LIN {X 0,Y 165.753,Z 434.239,A -85,B 0,C 180,E1 -23560.172,E2 -23560.172} C_VEL
LIN {X 0,Y 161.563,Z 431.762,A -85,B 0,C 180,E1 -23564.871,E2 -23564.871} C_VEL
LIN {X 0,Y 158.534,Z 427.948,A -85,B 0,C 180,E1 -23569.786,E2 -23569.786} C_VEL
LIN {X 0,Y 156.538,Z 422.635,A -85,B 0,C 180,E1 -23574.848,E2 -23574.848} C_VEL
LIN {X 0,Y 155.81,Z 417.574,A -85,B 0,C 180,E1 -23578.708,E2 -23578.708} C_VEL
LIN {X 0,Y 155.882,Z 410.304,A -85,B 0,C 180,E1 -23583.231,E2 -23583.231} C_VEL
LIN {X 0,Y 156.223,Z 402.738,A -85,B 0,C 180,E1 -23587.107,E2 -23587.107} C_VEL
LIN {X 0,Y 156.974,Z 393.545,A -85,B 0,C 180,E1 -23590.969,E2 -23590.969} C_VEL
LIN {X 0,Y 158.157,Z 382.372,A -85,B 0,C 180,E1 -23594.804,E2 -23594.804} C_VEL
LIN {X 0,Y 159.494,Z 371.159,A -85,B 0,C 180,E1 -23597.966,E2 -23597.966} C_VEL
LIN {X 0,Y 161.026,Z 358.78,A -85,B 0,C 180,E1 -23600.77,E2 -23600.77} C_VEL
LIN {X 0,Y 161.777,Z 350.482,A -85,B 0,C 180,E1 -23602.342,E2 -23602.342} C_VEL
LIN {X 0,Y 158.681,Z 336.403,A -85,B 0,C 180,E1 -23604.681,E2 -23604.681} C_VEL
LIN {X 0,Y 157.439,Z 330.353,A -85,B 0,C 180,E1 -23605.533,E2 -23605.533} C_VEL
LIN {X 0,Y 157.983,Z 332.419,A -85,B 0,C 180,E1 -23609.298,E2 -23609.298} C_VEL
LIN {X 0,Y 158.474,Z 334.327,A -85,B 0,C 180,E1 -23612.583,E2 -23612.583} C_VEL
LIN {X 0,Y 159.405,Z 337.957,A -85,B 0,C 180,E1 -23618.116,E2 -23618.116} C_VEL
LIN {X 0,Y 159.659,Z 338.968,A -85,B 0,C 180,E1 -23619.459,E2 -23619.459} C_VEL
LIN {X 0,Y 161.445,Z 342.254,A -85,B 0,C 180,E1 -23620.495,E2 -23620.495} C_VEL
LIN {X 0,Y 163.231,Z 344.63,A -85,B 0,C 180,E1 -23621.438,E2 -23621.438} C_VEL
LIN {X 0,Y 166.552,Z 350.082,A -85,B 0,C 180,E1 -23623.291,E2 -23623.291} C_VEL
LIN {X 0,Y 170.558,Z 357.475,A -85,B 0,C 180,E1 -23625.662,E2 -23625.662} C_VEL
LIN {X 0,Y 174.376,Z 366.782,A -85,B 0,C 180,E1 -23628.342,E2 -23628.342} C_VEL
LIN {X 0,Y 176.434,Z 377.226,A -85,B 0,C 180,E1 -23630.963,E2 -23630.963} C_VEL
LIN {X 0,Y 177.459,Z 387.081,A -85,B 0,C 180,E1 -23633.555,E2 -23633.555} C_VEL
LIN {X 0,Y 177.688,Z 393.471,A -85,B 0,C 180,E1 -23635.349,E2 -23635.349} C_VEL
LIN {X 0,Y 177.13,Z 395.819,A -85,B 0,C 180,E1 -23635.914,E2 -23635.914} C_VEL
LIN {X 0,Y 173.857,Z 405.236,A -85,B 0,C 180,E1 -23638.297,E2 -23638.297} C_VEL
LIN {X 0,Y 171.211,Z 412.228,A -85,B 0,C 180,E1 -23640.489,E2 -23640.489} C_VEL
LIN {X 0,Y 167.26,Z 420.911,A -85,B 0,C 180,E1 -23643.82,E2 -23643.82} C_VEL
LIN {X 0,Y 163.998,Z 427.85,A -85,B 0,C 180,E1 -23647.313,E2 -23647.313} C_VEL
LIN {X 0,Y 161.206,Z 433.361,A -85,B 0,C 180,E1 -23650.915,E2 -23650.915} C_VEL
LIN {X 0,Y 158.948,Z 437.681,A -85,B 0,C 180,E1 -23654.615,E2 -23654.615} C_VEL
LIN {X 0,Y 157.815,Z 439.949,A -85,B 0,C 180,E1 -23657.134,E2 -23657.134} C_VEL
LIN {X 0,Y 156.561,Z 442.532,A -85,B 0,C 180,E1 -23660.962,E2 -23660.962} C_VEL
LIN {X 0,Y 155.775,Z 444.181,A -85,B 0,C 180,E1 -23664.823,E2 -23664.823} C_VEL
LIN {X 0,Y 155.382,Z 445.015,A -85,B 0,C 180,E1 -23670,E2 -23670} C_VEL
LIN {X 0,Y 155.466,Z 444.818,A -85,B 0,C 180,E1 -23672.591,E2 -23672.591} C_VEL
LIN {X 0,Y 156.224,Z 443.266,A -85,B 0,C 180,E1 -23677.756,E2 -23677.756} C_VEL
LIN {X 0,Y 156.889,Z 441.903,A -85,B 0,C 180,E1 -23680.322,E2 -23680.322} C_VEL
LIN {X 0,Y 158.282,Z 439.04,A -85,B 0,C 180,E1 -23684.135,E2 -23684.135} C_VEL
LIN {X 0,Y 160.319,Z 435.137,A -85,B 0,C 180,E1 -23687.87,E2 -23687.87} C_VEL
LIN {X 0,Y 162.92,Z 430.072,A -85,B 0,C 180,E1 -23691.511,E2 -23691.511} C_VEL
LIN {X 0,Y 165.997,Z 423.682,A -85,B 0,C 180,E1 -23695.048,E2 -23695.048} C_VEL
LIN {X 0,Y 169.805,Z 415.717,A -85,B 0,C 180,E1 -23698.423,E2 -23698.423} C_VEL
LIN {X 0,Y 173.186,Z 407.595,A -85,B 0,C 180,E1 -23701.15,E2 -23701.15} C_VEL
LIN {X 0,Y 176.252,Z 398.682,A -85,B 0,C 180,E1 -23703.591,E2 -23703.591} C_VEL
LIN {X 0,Y 177.751,Z 394.094,A -85,B 0,C 180,E1 -23704.637,E2 -23704.637} C_VEL
LIN {X 0,Y 177.274,Z 383.59,A -85,B 0,C 180,E1 -23707.542,E2 -23707.542} C_VEL
LIN {X 0,Y 175.939,Z 373.719,A -85,B 0,C 180,E1 -23710.085,E2 -23710.085} C_VEL
LIN {X 0,Y 174.068,Z 365.643,A -85,B 0,C 180,E1 -23712.143,E2 -23712.143} C_VEL
LIN {X 0,Y 170.123,Z 356.525,A -85,B 0,C 180,E1 -23714.824,E2 -23714.824} C_VEL
LIN {X 0,Y 165.27,Z 347.901,A -85,B 0,C 180,E1 -23717.637,E2 -23717.637} C_VEL
LIN {X 0,Y 162.421,Z 343.392,A -85,B 0,C 180,E1 -23719.218,E2 -23719.218} C_VEL
LIN {X 0,Y 160.135,Z 340.062,A -85,B 0,C 180,E1 -23720.478,E2 -23720.478} C_VEL
LIN {X 0,Y 159.646,Z 338.902,A -85,B 0,C 180,E1 -23720.873,E2 -23720.873} C_VEL
LIN {X 0,Y 158.84,Z 336.211,A -85,B 0,C 180,E1 -23724.887,E2 -23724.887} C_VEL
LIN {X 0,Y 157.779,Z 334.62,A -85,B 0,C 180,E1 -23727.815,E2 -23727.815} C_VEL
LIN {X 0,Y 156.887,Z 333.987,A -85,B 0,C 180,E1 -23729.706,E2 -23729.706} C_VEL
LIN {X 0,Y 156.589,Z 338.43,A -85,B 0,C 180,E1 -23733.887,E2 -23733.887} C_VEL
LIN {X 0,Y 158.408,Z 353.582,A -85,B 0,C 180,E1 -23735.786,E2 -23735.786} C_VEL
LIN {X 0,Y 160.641,Z 367.663,A -85,B 0,C 180,E1 -23738.039,E2 -23738.039} C_VEL
LIN {X 0,Y 160.973,Z 370.884,A -85,B 0,C 180,E1 -23738.627,E2 -23738.627} C_VEL
LIN {X 0,Y 159.654,Z 382.742,A -85,B 0,C 180,E1 -23741.055,E2 -23741.055} C_VEL
LIN {X 0,Y 158.31,Z 393.87,A -85,B 0,C 180,E1 -23743.891,E2 -23743.891} C_VEL
LIN {X 0,Y 157.104,Z 404.147,A -85,B 0,C 180,E1 -23747.075,E2 -23747.075} C_VEL
LIN {X 0,Y 156.285,Z 412.837,A -85,B 0,C 180,E1 -23750.291,E2 -23750.291} C_VEL
LIN {X 0,Y 155.643,Z 421.458,A -85,B 0,C 180,E1 -23754.151,E2 -23754.151} C_VEL
LIN {X 0,Y 155.47,Z 428.59,A -85,B 0,C 180,E1 -23758.057,E2 -23758.057} C_VEL
LIN {X 0,Y 155.577,Z 435.33,A -85,B 0,C 180,E1 -23762.589,E2 -23762.589} C_VEL
LIN {X 0,Y 156.239,Z 439.911,A -85,B 0,C 180,E1 -23766.457,E2 -23766.457} C_VEL
LIN {X 0,Y 157.731,Z 444.459,A -85,B 0,C 180,E1 -23771.404,E2 -23771.404} C_VEL
LIN {X 0,Y 159.963,Z 447.144,A -85,B 0,C 180,E1 -23775.284,E2 -23775.284} C_VEL
LIN {X 0,Y 163.92,Z 449.371,A -85,B 0,C 180,E1 -23780.06,E2 -23780.06} C_VEL
LIN {X 0,Y 169.127,Z 450.293,A -85,B 0,C 180,E1 -23784.554,E2 -23784.554} C_VEL
LIN {X 0,Y 175.467,Z 449.904,A -85,B 0,C 180,E1 -23788.727,E2 -23788.727} C_VEL
LIN {X 0,Y 182.919,Z 448.24,A -85,B 0,C 180,E1 -23792.541,E2 -23792.541} C_VEL
LIN {X 0,Y 191.342,Z 445.326,A -85,B 0,C 180,E1 -23795.993,E2 -23795.993} C_VEL
LIN {X 0,Y 200.7,Z 441.045,A -85,B 0,C 180,E1 -23799.073,E2 -23799.073} C_VEL
LIN {X 0,Y 210.694,Z 435.47,A -85,B 0,C 180,E1 -23801.846,E2 -23801.846} C_VEL
LIN {X 0,Y 211.205,Z 435.279,A -85,B 0,C 180,E1 -23802.94,E2 -23802.94} C_VEL
LIN {X 0,Y 210.36,Z 436.026,A -85,B 0,C 180,E1 -23804.085,E2 -23804.085} C_VEL
LIN {X 0,Y 206.003,Z 439.07,A -85,B 0,C 180,E1 -23805.623,E2 -23805.623} C_VEL
LIN {X 0,Y 194.505,Z 446.435,A -85,B 0,C 180,E1 -23809.429,E2 -23809.429} C_VEL
LIN {X 0,Y 185.399,Z 451.418,A -85,B 0,C 180,E1 -23812.662,E2 -23812.662} C_VEL
LIN {X 0,Y 177.209,Z 455.306,A -85,B 0,C 180,E1 -23816.273,E2 -23816.273} C_VEL
LIN {X 0,Y 170.283,Z 458.104,A -85,B 0,C 180,E1 -23820.312,E2 -23820.312} C_VEL
LIN {X 0,Y 164.595,Z 459.85,A -85,B 0,C 180,E1 -23824.723,E2 -23824.723} C_VEL
LIN {X 0,Y 160.207,Z 460.514,A -85,B 0,C 180,E1 -23829.455,E2 -23829.455} C_VEL
LIN {X 0,Y 157.293,Z 460.078,A -85,B 0,C 180,E1 -23834.45,E2 -23834.45} C_VEL
LIN {X 0,Y 156.148,Z 459.074,A -85,B 0,C 180,E1 -23838.479,E2 -23838.479} C_VEL
LIN {X 0,Y 155.39,Z 461.312,A -85,B 0,C 180,E1 -23842.202,E2 -23842.202} C_VEL
LIN {X 0,Y 155.146,Z 462.974,A -85,B 0,C 180,E1 -23847.404,E2 -23847.404} C_VEL
LIN {X 0,Y 155.383,Z 463.209,A -85,B 0,C 180,E1 -23850,E2 -23850} C_VEL
LIN {X 0,Y 155.08,Z 462.56,A -85,B 0,C 180,E1 -23854.433,E2 -23854.433} C_VEL
LIN {X 0,Y 155.153,Z 461.271,A -85,B 0,C 180,E1 -23857.81,E2 -23857.81} C_VEL
LIN {X 0,Y 155.501,Z 459.802,A -85,B 0,C 180,E1 -23860.415,E2 -23860.415} C_VEL
LIN {X 0,Y 156.455,Z 456.851,A -85,B 0,C 180,E1 -23864.204,E2 -23864.204} C_VEL
LIN {X 0,Y 156.313,Z 455.572,A -85,B 0,C 180,E1 -23865.589,E2 -23865.589} C_VEL
LIN {X 0,Y 153.093,Z 451.08,A -85,B 0,C 180,E1 -23870.172,E2 -23870.172} C_VEL
LIN {X 0,Y 153.396,Z 450.467,A -85,B 0,C 180,E1 -23871.636,E2 -23871.636} C_VEL
LIN {X 0,Y 157.584,Z 449.759,A -85,B 0,C 180,E1 -23876.486,E2 -23876.486} C_VEL
LIN {X 0,Y 163.273,Z 448.055,A -85,B 0,C 180,E1 -23881.1,E2 -23881.1} C_VEL
LIN {X 0,Y 170.372,Z 445.383,A -85,B 0,C 180,E1 -23885.276,E2 -23885.276} C_VEL
LIN {X 0,Y 178.668,Z 441.731,A -85,B 0,C 180,E1 -23889.004,E2 -23889.004} C_VEL
LIN {X 0,Y 189.566,Z 435.946,A -85,B 0,C 180,E1 -23893.305,E2 -23893.305} C_VEL
LIN {X 0,Y 193.556,Z 433.494,A -85,B 0,C 180,E1 -23895.076,E2 -23895.076} C_VEL
LIN {X 0,Y 195.412,Z 432.26,A -85,B 0,C 180,E1 -23895.997,E2 -23895.997} C_VEL
LIN {X 0,Y 197.524,Z 430.74,A -85,B 0,C 180,E1 -23897.466,E2 -23897.466} C_VEL
LIN {X 0,Y 197.825,Z 430.354,A -85,B 0,C 180,E1 -23898.25,E2 -23898.25} C_VEL
LIN {X 0,Y 198.082,Z 429.735,A -85,B 0,C 180,E1 -23900.309,E2 -23900.309} C_VEL
LIN {X 0,Y 188.461,Z 433.218,A -85,B 0,C 180,E1 -23903.369,E2 -23903.369} C_VEL
LIN {X 0,Y 179.669,Z 435.441,A -85,B 0,C 180,E1 -23906.796,E2 -23906.796} C_VEL
LIN {X 0,Y 171.721,Z 436.42,A -85,B 0,C 180,E1 -23910.586,E2 -23910.586} C_VEL
LIN {X 0,Y 164.78,Z 436.179,A -85,B 0,C 180,E1 -23914.754,E2 -23914.754} C_VEL
LIN {X 0,Y 159.11,Z 434.652,A -85,B 0,C 180,E1 -23919.307,E2 -23919.307} C_VEL
LIN {X 0,Y 154.737,Z 431.839,A -85,B 0,C 180,E1 -23924.186,E2 -23924.186} C_VEL
LIN {X 0,Y 151.567,Z 427.625,A -85,B 0,C 180,E1 -23929.311,E2 -23929.311} C_VEL
LIN {X 0,Y 149.492,Z 421.939,A -85,B 0,C 180,E1 -23934.605,E2 -23934.605} C_VEL
LIN {X 0,Y 148.727,Z 414.582,A -85,B 0,C 180,E1 -23940,E2 -23940} C_VEL
LIN {X 0,Y 149.03,Z 406.5,A -85,B 0,C 180,E1 -23944.734,E2 -23944.734} C_VEL
LIN {X 0,Y 149.553,Z 396.83,A -85,B 0,C 180,E1 -23949.297,E2 -23949.297} C_VEL
LIN {X 0,Y 150.411,Z 387.773,A -85,B 0,C 180,E1 -23952.824,E2 -23952.824} C_VEL
LIN {X 0,Y 151.711,Z 376.334,A -85,B 0,C 180,E1 -23956.484,E2 -23956.484} C_VEL
LIN {X 0,Y 153.302,Z 363.69,A -85,B 0,C 180,E1 -23959.761,E2 -23959.761} C_VEL
LIN {X 0,Y 154.707,Z 352.272,A -85,B 0,C 180,E1 -23962.167,E2 -23962.167} C_VEL
LIN {X 0,Y 152.905,Z 343.422,A -85,B 0,C 180,E1 -23963.779,E2 -23963.779} C_VEL
LIN {X 0,Y 150.839,Z 333.597,A -85,B 0,C 180,E1 -23965.402,E2 -23965.402} C_VEL
LIN {X 0,Y 151.352,Z 334.822,A -85,B 0,C 180,E1 -23968.083,E2 -23968.083} C_VEL
LIN {X 0,Y 152.138,Z 337.991,A -85,B 0,C 180,E1 -23973.746,E2 -23973.746} C_VEL
LIN {X 0,Y 152.527,Z 339.479,A -85,B 0,C 180,E1 -23976.08,E2 -23976.08} C_VEL
LIN {X 0,Y 154.477,Z 342.78,A -85,B 0,C 180,E1 -23977.367,E2 -23977.367} C_VEL
LIN {X 0,Y 156.395,Z 345.088,A -85,B 0,C 180,E1 -23978.51,E2 -23978.51} C_VEL
LIN {X 0,Y 158.911,Z 349.057,A -85,B 0,C 180,E1 -23980.094,E2 -23980.094} C_VEL
LIN {X 0,Y 162.644,Z 355.633,A -85,B 0,C 180,E1 -23982.5,E2 -23982.5} C_VEL
LIN {X 0,Y 166.311,Z 363.122,A -85,B 0,C 180,E1 -23985.059,E2 -23985.059} C_VEL
LIN {X 0,Y 169.218,Z 370.991,A -85,B 0,C 180,E1 -23987.494,E2 -23987.494} C_VEL
LIN {X 0,Y 170.838,Z 380.954,A -85,B 0,C 180,E1 -23990.188,E2 -23990.188} C_VEL
LIN {X 0,Y 171.504,Z 390.512,A -85,B 0,C 180,E1 -23992.898,E2 -23992.898} C_VEL
LIN {X 0,Y 171.539,Z 395.184,A -85,B 0,C 180,E1 -23994.308,E2 -23994.308} C_VEL
LIN {X 0,Y 167.86,Z 405.647,A -85,B 0,C 180,E1 -23997.024,E2 -23997.024} C_VEL
LIN {X 0,Y 165.094,Z 412.639,A -85,B 0,C 180,E1 -23999.28,E2 -23999.28} C_VEL
LIN {X 0,Y 160.935,Z 421.324,A -85,B 0,C 180,E1 -24002.707,E2 -24002.707} C_VEL
LIN {X 0,Y 157.48,Z 428.265,A -85,B 0,C 180,E1 -24006.318,E2 -24006.318} C_VEL
LIN {X 0,Y 154.521,Z 433.776,A -85,B 0,C 180,E1 -24010.055,E2 -24010.055} C_VEL
LIN {X 0,Y 152.12,Z 438.097,A -85,B 0,C 180,E1 -24013.907,E2 -24013.907} C_VEL
LIN {X 0,Y 150.921,Z 440.363,A -85,B 0,C 180,E1 -24016.536,E2 -24016.536} C_VEL
LIN {X 0,Y 149.496,Z 443.105,A -85,B 0,C 180,E1 -24020.838,E2 -24020.838} C_VEL
LIN {X 0,Y 148.726,Z 444.595,A -85,B 0,C 180,E1 -24024.577,E2 -24024.577} C_VEL
LIN {X 0,Y 148.301,Z 445.43,A -85,B 0,C 180,E1 -24030,E2 -24030} C_VEL
LIN {X 0,Y 148.393,Z 445.232,A -85,B 0,C 180,E1 -24032.715,E2 -24032.715} C_VEL
LIN {X 0,Y 149.215,Z 443.68,A -85,B 0,C 180,E1 -24038.123,E2 -24038.123} C_VEL
LIN {X 0,Y 149.915,Z 442.318,A -85,B 0,C 180,E1 -24040.808,E2 -24040.808} C_VEL
LIN {X 0,Y 151.425,Z 439.453,A -85,B 0,C 180,E1 -24044.79,E2 -24044.79} C_VEL
LIN {X 0,Y 153.582,Z 435.55,A -85,B 0,C 180,E1 -24048.683,E2 -24048.683} C_VEL
LIN {X 0,Y 156.353,Z 430.482,A -85,B 0,C 180,E1 -24052.462,E2 -24052.462} C_VEL
LIN {X 0,Y 159.6,Z 424.092,A -85,B 0,C 180,E1 -24056.126,E2 -24056.126} C_VEL
LIN {X 0,Y 163.622,Z 416.123,A -85,B 0,C 180,E1 -24059.601,E2 -24059.601} C_VEL
LIN {X 0,Y 167.108,Z 408.095,A -85,B 0,C 180,E1 -24062.379,E2 -24062.379} C_VEL
LIN {X 0,Y 170.363,Z 399.191,A -85,B 0,C 180,E1 -24064.881,E2 -24064.881} C_VEL
LIN {X 0,Y 171.58,Z 395.68,A -85,B 0,C 180,E1 -24065.704,E2 -24065.704} C_VEL
LIN {X 0,Y 171.41,Z 386.763,A -85,B 0,C 180,E1 -24068.346,E2 -24068.346} C_VEL
LIN {X 0,Y 170.239,Z 375.936,A -85,B 0,C 180,E1 -24071.341,E2 -24071.341} C_VEL
LIN {X 0,Y 168.776,Z 369.321,A -85,B 0,C 180,E1 -24073.167,E2 -24073.167} C_VEL
LIN {X 0,Y 165.587,Z 361.345,A -85,B 0,C 180,E1 -24075.718,E2 -24075.718} C_VEL
LIN {X 0,Y 161.339,Z 353.166,A -85,B 0,C 180,E1 -24078.58,E2 -24078.58} C_VEL
LIN {X 0,Y 158.362,Z 348.322,A -85,B 0,C 180,E1 -24080.463,E2 -24080.463} C_VEL
LIN {X 0,Y 155.848,Z 344.352,A -85,B 0,C 180,E1 -24082.055,E2 -24082.055} C_VEL
LIN {X 0,Y 152.98,Z 340.619,A -85,B 0,C 180,E1 -24083.839,E2 -24083.839} C_VEL
LIN {X 0,Y 152.449,Z 339.441,A -85,B 0,C 180,E1 -24084.305,E2 -24084.305} C_VEL
LIN {X 0,Y 151.762,Z 338.268,A -85,B 0,C 180,E1 -24086.468,E2 -24086.468} C_VEL
LIN {X 0,Y 150.617,Z 337.054,A -85,B 0,C 180,E1 -24089.117,E2 -24089.117} C_VEL
LIN {X 0,Y 149.674,Z 336.321,A -85,B 0,C 180,E1 -24091.23,E2 -24091.23} C_VEL
LIN {X 0,Y 149.517,Z 338.899,A -85,B 0,C 180,E1 -24093.734,E2 -24093.734} C_VEL
LIN {X 0,Y 151.314,Z 354.037,A -85,B 0,C 180,E1 -24095.692,E2 -24095.692} C_VEL
LIN {X 0,Y 153.57,Z 368.285,A -85,B 0,C 180,E1 -24098.077,E2 -24098.077} C_VEL
LIN {X 0,Y 153.869,Z 370.852,A -85,B 0,C 180,E1 -24098.567,E2 -24098.567} C_VEL
LIN {X 0,Y 152.513,Z 382.915,A -85,B 0,C 180,E1 -24101.181,E2 -24101.181} C_VEL
LIN {X 0,Y 151,Z 395.136,A -85,B 0,C 180,E1 -24104.477,E2 -24104.477} C_VEL
LIN {X 0,Y 149.868,Z 405.309,A -85,B 0,C 180,E1 -24107.817,E2 -24107.817} C_VEL
LIN {X 0,Y 149.094,Z 413.784,A -85,B 0,C 180,E1 -24111.188,E2 -24111.188} C_VEL
LIN {X 0,Y 148.566,Z 422.244,A -85,B 0,C 180,E1 -24115.251,E2 -24115.251} C_VEL
LIN {X 0,Y 148.463,Z 429.301,A -85,B 0,C 180,E1 -24119.322,E2 -24119.322} C_VEL
LIN {X 0,Y 148.76,Z 435.899,A -85,B 0,C 180,E1 -24124.064,E2 -24124.064} C_VEL
LIN {X 0,Y 149.57,Z 440.46,A -85,B 0,C 180,E1 -24128.104,E2 -24128.104} C_VEL
LIN {X 0,Y 151.519,Z 445.084,A -85,B 0,C 180,E1 -24133.41,E2 -24133.41} C_VEL
LIN {X 0,Y 155.053,Z 448.373,A -85,B 0,C 180,E1 -24138.499,E2 -24138.499} C_VEL
LIN {X 0,Y 159.788,Z 450.348,A -85,B 0,C 180,E1 -24143.319,E2 -24143.319} C_VEL
LIN {X 0,Y 165.848,Z 451,A -85,B 0,C 180,E1 -24147.784,E2 -24147.784} C_VEL
LIN {X 0,Y 173.102,Z 450.409,A -85,B 0,C 180,E1 -24151.857,E2 -24151.857} C_VEL
LIN {X 0,Y 181.833,Z 448.487,A -85,B 0,C 180,E1 -24155.74,E2 -24155.74} C_VEL
LIN {X 0,Y 190.575,Z 445.528,A -85,B 0,C 180,E1 -24158.824,E2 -24158.824} C_VEL
LIN {X 0,Y 200.582,Z 441.177,A -85,B 0,C 180,E1 -24161.738,E2 -24161.738} C_VEL
LIN {X 0,Y 204.307,Z 439.31,A -85,B 0,C 180,E1 -24162.7,E2 -24162.7} C_VEL
LIN {X 0,Y 203.582,Z 439.873,A -85,B 0,C 180,E1 -24163.534,E2 -24163.534} C_VEL
LIN {X 0,Y 191.618,Z 446.746,A -85,B 0,C 180,E1 -24167.271,E2 -24167.271} C_VEL
LIN {X 0,Y 183.001,Z 451.032,A -85,B 0,C 180,E1 -24170.182,E2 -24170.182} C_VEL
LIN {X 0,Y 175.486,Z 454.225,A -85,B 0,C 180,E1 -24173.077,E2 -24173.077} C_VEL
LIN {X 0,Y 167.006,Z 457.295,A -85,B 0,C 180,E1 -24177.315,E2 -24177.315} C_VEL
LIN {X 0,Y 161.028,Z 458.939,A -85,B 0,C 180,E1 -24181.309,E2 -24181.309} C_VEL
LIN {X 0,Y 155.691,Z 459.759,A -85,B 0,C 180,E1 -24186.029,E2 -24186.029} C_VEL
LIN {X 0,Y 151.805,Z 459.525,A -85,B 0,C 180,E1 -24191.09,E2 -24191.09} C_VEL
LIN {X 0,Y 149.455,Z 458.077,A -85,B 0,C 180,E1 -24197.093,E2 -24197.093} C_VEL
LIN {X 0,Y 148.349,Z 460.897,A -85,B 0,C 180,E1 -24201.829,E2 -24201.829} C_VEL
LIN {X 0,Y 148.068,Z 462.178,A -85,B 0,C 180,E1 -24205.387,E2 -24205.387} C_VEL
LIN {X 0,Y 148.29,Z 462.794,A -85,B 0,C 180,E1 -24210,E2 -24210} C_VEL
LIN {X 0,Y 148.01,Z 462.237,A -85,B 0,C 180,E1 -24214.328,E2 -24214.328} C_VEL
LIN {X 0,Y 148.084,Z 460.853,A -85,B 0,C 180,E1 -24218.186,E2 -24218.186} C_VEL
LIN {X 0,Y 148.497,Z 459.384,A -85,B 0,C 180,E1 -24220.913,E2 -24220.913} C_VEL
LIN {X 0,Y 149.591,Z 456.351,A -85,B 0,C 180,E1 -24224.975,E2 -24224.975} C_VEL
LIN {X 0,Y 151.576,Z 452.267,A -85,B 0,C 180,E1 -24228.939,E2 -24228.939} C_VEL
LIN {X 0,Y 152.564,Z 450.503,A -85,B 0,C 180,E1 -24230.388,E2 -24230.388} C_VEL
LIN {X 0,Y 153.396,Z 450.467,A -85,B 0,C 180,E1 -24231.636,E2 -24231.636} C_VEL
LIN {X 0,Y 154.375,Z 450.218,A -85,B 0,C 180,E1 -24233.806,E2 -24233.806} C_VEL
LIN {X 0,Y 155.587,Z 448.449,A -85,B 0,C 180,E1 -24240.363,E2 -24240.363} C_VEL
LIN {X 0,Y 157.292,Z 447.668,A -85,B 0,C 180,E1 -24242.407,E2 -24242.407} C_VEL
LIN {X 0,Y 158.172,Z 447.386,A -85,B 0,C 180,E1 -24243.036,E2 -24243.036} C_VEL
LIN {X 0,Y 164.638,Z 445.411,A -85,B 0,C 180,E1 -24246.7,E2 -24246.7} C_VEL
LIN {X 0,Y 173.226,Z 442.231,A -85,B 0,C 180,E1 -24250.477,E2 -24250.477} C_VEL
LIN {X 0,Y 184.514,Z 437.059,A -85,B 0,C 180,E1 -24254.802,E2 -24254.802} C_VEL
LIN {X 0,Y 188.637,Z 434.859,A -85,B 0,C 180,E1 -24256.595,E2 -24256.595} C_VEL
LIN {X 0,Y 190.392,Z 433.799,A -85,B 0,C 180,E1 -24257.584,E2 -24257.584} C_VEL
LIN {X 0,Y 191.359,Z 433.091,A -85,B 0,C 180,E1 -24258.617,E2 -24258.617} C_VEL
LIN {X 0,Y 190.438,Z 433.174,A -85,B 0,C 180,E1 -24259.772,E2 -24259.772} C_VEL
LIN {X 0,Y 183.02,Z 435.254,A -85,B 0,C 180,E1 -24262.091,E2 -24262.091} C_VEL
LIN {X 0,Y 173.918,Z 436.996,A -85,B 0,C 180,E1 -24265.546,E2 -24265.546} C_VEL
LIN {X 0,Y 165.647,Z 437.572,A -85,B 0,C 180,E1 -24269.394,E2 -24269.394} C_VEL
LIN {X 0,Y 158.429,Z 436.887,A -85,B 0,C 180,E1 -24273.666,E2 -24273.666} C_VEL
LIN {X 0,Y 152.509,Z 434.941,A -85,B 0,C 180,E1 -24278.367,E2 -24278.367} C_VEL
LIN {X 0,Y 147.938,Z 431.727,A -85,B 0,C 180,E1 -24283.439,E2 -24283.439} C_VEL
LIN {X 0,Y 144.614,Z 427.179,A -85,B 0,C 180,E1 -24288.791,E2 -24288.791} C_VEL
LIN {X 0,Y 142.462,Z 421.11,A -85,B 0,C 180,E1 -24294.338,E2 -24294.338} C_VEL
LIN {X 0,Y 141.71,Z 413.335,A -85,B 0,C 180,E1 -24300,E2 -24300} C_VEL
LIN {X 0,Y 142.023,Z 404.891,A -85,B 0,C 180,E1 -24304.968,E2 -24304.968} C_VEL
LIN {X 0,Y 142.529,Z 395.794,A -85,B 0,C 180,E1 -24309.293,E2 -24309.293} C_VEL
LIN {X 0,Y 143.579,Z 385.207,A -85,B 0,C 180,E1 -24313.445,E2 -24313.445} C_VEL
LIN {X 0,Y 144.969,Z 373.249,A -85,B 0,C 180,E1 -24317.274,E2 -24317.274} C_VEL
LIN {X 0,Y 146.487,Z 361.182,A -85,B 0,C 180,E1 -24320.355,E2 -24320.355} C_VEL
LIN {X 0,Y 147.48,Z 353.393,A -85,B 0,C 180,E1 -24322.042,E2 -24322.042} C_VEL
LIN {X 0,Y 147.488,Z 351.505,A -85,B 0,C 180,E1 -24322.409,E2 -24322.409} C_VEL
LIN {X 0,Y 144.535,Z 338.06,A -85,B 0,C 180,E1 -24324.854,E2 -24324.854} C_VEL
LIN {X 0,Y 144.246,Z 336.748,A -85,B 0,C 180,E1 -24325.127,E2 -24325.127} C_VEL
LIN {X 0,Y 144.643,Z 336.965,A -85,B 0,C 180,E1 -24325.932,E2 -24325.932} C_VEL
LIN {X 0,Y 145.352,Z 339.638,A -85,B 0,C 180,E1 -24331.317,E2 -24331.317} C_VEL
LIN {X 0,Y 145.559,Z 340.272,A -85,B 0,C 180,E1 -24332.149,E2 -24332.149} C_VEL
LIN {X 0,Y 147.748,Z 343.714,A -85,B 0,C 180,E1 -24333.845,E2 -24333.845} C_VEL
LIN {X 0,Y 149.613,Z 345.751,A -85,B 0,C 180,E1 -24335.131,E2 -24335.131} C_VEL
LIN {X 0,Y 152.192,Z 349.675,A -85,B 0,C 180,E1 -24336.997,E2 -24336.997} C_VEL
LIN {X 0,Y 156.002,Z 356.166,A -85,B 0,C 180,E1 -24339.765,E2 -24339.765} C_VEL
LIN {X 0,Y 158.485,Z 360.883,A -85,B 0,C 180,E1 -24341.638,E2 -24341.638} C_VEL
LIN {X 0,Y 161.539,Z 367.596,A -85,B 0,C 180,E1 -24344.116,E2 -24344.116} C_VEL
LIN {X 0,Y 163.836,Z 374.444,A -85,B 0,C 180,E1 -24346.422,E2 -24346.422} C_VEL
LIN {X 0,Y 165.028,Z 383.315,A -85,B 0,C 180,E1 -24349.002,E2 -24349.002} C_VEL
LIN {X 0,Y 165.477,Z 392.709,A -85,B 0,C 180,E1 -24351.86,E2 -24351.86} C_VEL
LIN {X 0,Y 165.46,Z 395.829,A -85,B 0,C 180,E1 -24352.854,E2 -24352.854} C_VEL
LIN {X 0,Y 164.733,Z 398.923,A -85,B 0,C 180,E1 -24353.705,E2 -24353.705} C_VEL
LIN {X 0,Y 161.579,Z 407.086,A -85,B 0,C 180,E1 -24355.975,E2 -24355.975} C_VEL
LIN {X 0,Y 158.273,Z 414.645,A -85,B 0,C 180,E1 -24358.55,E2 -24358.55} C_VEL
LIN {X 0,Y 154.681,Z 421.737,A -85,B 0,C 180,E1 -24361.505,E2 -24361.505} C_VEL
LIN {X 0,Y 151.025,Z 428.678,A -85,B 0,C 180,E1 -24365.24,E2 -24365.24} C_VEL
LIN {X 0,Y 147.867,Z 434.192,A -85,B 0,C 180,E1 -24369.116,E2 -24369.116} C_VEL
LIN {X 0,Y 145.33,Z 438.511,A -85,B 0,C 180,E1 -24373.133,E2 -24373.133} C_VEL
LIN {X 0,Y 144.024,Z 440.779,A -85,B 0,C 180,E1 -24375.878,E2 -24375.878} C_VEL
LIN {X 0,Y 142.376,Z 443.75,A -85,B 0,C 180,E1 -24380.841,E2 -24380.841} C_VEL
LIN {X 0,Y 141.681,Z 445.01,A -85,B 0,C 180,E1 -24384.306,E2 -24384.306} C_VEL
LIN {X 0,Y 141.221,Z 445.844,A -85,B 0,C 180,E1 -24390,E2 -24390} C_VEL
LIN {X 0,Y 141.322,Z 445.646,A -85,B 0,C 180,E1 -24392.851,E2 -24392.851} C_VEL
LIN {X 0,Y 141.658,Z 445.059,A -85,B 0,C 180,E1 -24395.695,E2 -24395.695} C_VEL
LIN {X 0,Y 142.32,Z 443.9,A -85,B 0,C 180,E1 -24399.018,E2 -24399.018} C_VEL
LIN {X 0,Y 143.972,Z 440.909,A -85,B 0,C 180,E1 -24404.127,E2 -24404.127} C_VEL
LIN {X 0,Y 146.041,Z 437.362,A -85,B 0,C 180,E1 -24408.228,E2 -24408.228} C_VEL
LIN {X 0,Y 148.809,Z 432.697,A -85,B 0,C 180,E1 -24412.199,E2 -24412.199} C_VEL
LIN {X 0,Y 152.094,Z 426.782,A -85,B 0,C 180,E1 -24416.039,E2 -24416.039} C_VEL
LIN {X 0,Y 156.014,Z 419.406,A -85,B 0,C 180,E1 -24419.704,E2 -24419.704} C_VEL
LIN {X 0,Y 160.277,Z 410.568,A -85,B 0,C 180,E1 -24423.046,E2 -24423.046} C_VEL
LIN {X 0,Y 164.15,Z 400.747,A -85,B 0,C 180,E1 -24425.989,E2 -24425.989} C_VEL
LIN {X 0,Y 165.447,Z 397.325,A -85,B 0,C 180,E1 -24426.83,E2 -24426.83} C_VEL
LIN {X 0,Y 165.483,Z 388.614,A -85,B 0,C 180,E1 -24429.572,E2 -24429.572} C_VEL
LIN {X 0,Y 164.566,Z 378.245,A -85,B 0,C 180,E1 -24432.641,E2 -24432.641} C_VEL
LIN {X 0,Y 163.095,Z 371.63,A -85,B 0,C 180,E1 -24434.683,E2 -24434.683} C_VEL
LIN {X 0,Y 159.337,Z 362.386,A -85,B 0,C 180,E1 -24437.969,E2 -24437.969} C_VEL
LIN {X 0,Y 154.999,Z 354.231,A -85,B 0,C 180,E1 -24441.223,E2 -24441.223} C_VEL
LIN {X 0,Y 152.226,Z 349.783,A -85,B 0,C 180,E1 -24443.22,E2 -24443.22} C_VEL
LIN {X 0,Y 149.553,Z 345.761,A -85,B 0,C 180,E1 -24445.161,E2 -24445.161} C_VEL
LIN {X 0,Y 144.999,Z 341.313,A -85,B 0,C 180,E1 -24448.394,E2 -24448.394} C_VEL
LIN {X 0,Y 144.105,Z 340.105,A -85,B 0,C 180,E1 -24449.197,E2 -24449.197} C_VEL
LIN {X 0,Y 142.483,Z 338.783,A -85,B 0,C 180,E1 -24453.058,E2 -24453.058} C_VEL
LIN {X 0,Y 142.463,Z 339.271,A -85,B 0,C 180,E1 -24453.543,E2 -24453.543} C_VEL
LIN {X 0,Y 144.249,Z 354.689,A -85,B 0,C 180,E1 -24455.673,E2 -24455.673} C_VEL
LIN {X 0,Y 146.501,Z 368.875,A -85,B 0,C 180,E1 -24458.174,E2 -24458.174} C_VEL
LIN {X 0,Y 146.564,Z 372.559,A -85,B 0,C 180,E1 -24458.922,E2 -24458.922} C_VEL
LIN {X 0,Y 145.216,Z 384.396,A -85,B 0,C 180,E1 -24461.664,E2 -24461.664} C_VEL
LIN {X 0,Y 143.717,Z 396.351,A -85,B 0,C 180,E1 -24465.123,E2 -24465.123} C_VEL
LIN {X 0,Y 142.718,Z 406.264,A -85,B 0,C 180,E1 -24468.64,E2 -24468.64} C_VEL
LIN {X 0,Y 141.828,Z 416.449,A -85,B 0,C 180,E1 -24473.056,E2 -24473.056} C_VEL
LIN {X 0,Y 141.518,Z 424.246,A -85,B 0,C 180,E1 -24477.153,E2 -24477.153} C_VEL
LIN {X 0,Y 141.515,Z 430.893,A -85,B 0,C 180,E1 -24481.423,E2 -24481.423} C_VEL
LIN {X 0,Y 142.032,Z 436.439,A -85,B 0,C 180,E1 -24485.679,E2 -24485.679} C_VEL
LIN {X 0,Y 143.412,Z 442.178,A -85,B 0,C 180,E1 -24491.304,E2 -24491.304} C_VEL
LIN {X 0,Y 146.352,Z 446.533,A -85,B 0,C 180,E1 -24496.746,E2 -24496.746} C_VEL
LIN {X 0,Y 150.689,Z 449.519,A -85,B 0,C 180,E1 -24501.908,E2 -24501.908} C_VEL
LIN {X 0,Y 156.38,Z 451.214,A -85,B 0,C 180,E1 -24506.706,E2 -24506.706} C_VEL
LIN {X 0,Y 163.27,Z 451.693,A -85,B 0,C 180,E1 -24511.101,E2 -24511.101} C_VEL
LIN {X 0,Y 171.344,Z 450.964,A -85,B 0,C 180,E1 -24515.046,E2 -24515.046} C_VEL
LIN {X 0,Y 180.363,Z 449.016,A -85,B 0,C 180,E1 -24518.569,E2 -24518.569} C_VEL
LIN {X 0,Y 190.352,Z 445.831,A -85,B 0,C 180,E1 -24521.65,E2 -24521.65} C_VEL
LIN {X 0,Y 195.591,Z 443.791,A -85,B 0,C 180,E1 -24523.056,E2 -24523.056} C_VEL
LIN {X 0,Y 184.148,Z 449.308,A -85,B 0,C 180,E1 -24526.609,E2 -24526.609} C_VEL
LIN {X 0,Y 174.41,Z 453.21,A -85,B 0,C 180,E1 -24529.854,E2 -24529.854} C_VEL
LIN {X 0,Y 165.616,Z 456.124,A -85,B 0,C 180,E1 -24533.552,E2 -24533.552} C_VEL
LIN {X 0,Y 158.103,Z 458.033,A -85,B 0,C 180,E1 -24537.763,E2 -24537.763} C_VEL
LIN {X 0,Y 151.888,Z 458.967,A -85,B 0,C 180,E1 -24542.438,E2 -24542.438} C_VEL
LIN {X 0,Y 147.034,Z 458.888,A -85,B 0,C 180,E1 -24547.518,E2 -24547.518} C_VEL
LIN {X 0,Y 143.784,Z 457.798,A -85,B 0,C 180,E1 -24552.946,E2 -24552.946} C_VEL
LIN {X 0,Y 142.886,Z 456.993,A -85,B 0,C 180,E1 -24555.581,E2 -24555.581} C_VEL
LIN {X 0,Y 141.875,Z 459.035,A -85,B 0,C 180,E1 -24558.571,E2 -24558.571} C_VEL
LIN {X 0,Y 141.305,Z 460.481,A -85,B 0,C 180,E1 -24561.419,E2 -24561.419} C_VEL
LIN {X 0,Y 140.972,Z 462.143,A -85,B 0,C 180,E1 -24567.142,E2 -24567.142} C_VEL
LIN {X 0,Y 141.199,Z 462.379,A -85,B 0,C 180,E1 -24570,E2 -24570} C_VEL
LIN {X 0,Y 140.929,Z 461.902,A -85,B 0,C 180,E1 -24574.147,E2 -24574.147} C_VEL
LIN {X 0,Y 141.037,Z 460.436,A -85,B 0,C 180,E1 -24578.598,E2 -24578.598} C_VEL
LIN {X 0,Y 141.483,Z 458.965,A -85,B 0,C 180,E1 -24581.461,E2 -24581.461} C_VEL
LIN {X 0,Y 142.696,Z 455.932,A -85,B 0,C 180,E1 -24585.717,E2 -24585.717} C_VEL
LIN {X 0,Y 144.879,Z 451.852,A -85,B 0,C 180,E1 -24589.851,E2 -24589.851} C_VEL
LIN {X 0,Y 146.419,Z 449.347,A -85,B 0,C 180,E1 -24592.024,E2 -24592.024} C_VEL
LIN {X 0,Y 151.274,Z 448.981,A -85,B 0,C 180,E1 -24597.684,E2 -24597.684} C_VEL
LIN {X 0,Y 158.172,Z 447.386,A -85,B 0,C 180,E1 -24603.036,E2 -24603.036} C_VEL
LIN {X 0,Y 160.624,Z 446.532,A -85,B 0,C 180,E1 -24604.938,E2 -24604.938} C_VEL
LIN {X 0,Y 166.25,Z 443.397,A -85,B 0,C 180,E1 -24610.765,E2 -24610.765} C_VEL
LIN {X 0,Y 169.073,Z 442.141,A -85,B 0,C 180,E1 -24612.482,E2 -24612.482} C_VEL
LIN {X 0,Y 170.248,Z 441.686,A -85,B 0,C 180,E1 -24612.993,E2 -24612.993} C_VEL
LIN {X 0,Y 179.576,Z 437.989,A -85,B 0,C 180,E1 -24616.388,E2 -24616.388} C_VEL
LIN {X 0,Y 183.13,Z 436.352,A -85,B 0,C 180,E1 -24617.901,E2 -24617.901} C_VEL
LIN {X 0,Y 183.921,Z 435.822,A -85,B 0,C 180,E1 -24618.809,E2 -24618.809} C_VEL
LIN {X 0,Y 172.801,Z 437.947,A -85,B 0,C 180,E1 -24622.406,E2 -24622.406} C_VEL
LIN {X 0,Y 163.797,Z 438.631,A -85,B 0,C 180,E1 -24626.097,E2 -24626.097} C_VEL
LIN {X 0,Y 155.711,Z 438.151,A -85,B 0,C 180,E1 -24630.232,E2 -24630.232} C_VEL
LIN {X 0,Y 148.894,Z 436.43,A -85,B 0,C 180,E1 -24634.861,E2 -24634.861} C_VEL
LIN {X 0,Y 143.386,Z 433.459,A -85,B 0,C 180,E1 -24639.934,E2 -24639.934} C_VEL
LIN {X 0,Y 139.257,Z 429.186,A -85,B 0,C 180,E1 -24645.384,E2 -24645.384} C_VEL
LIN {X 0,Y 136.392,Z 423.527,A -85,B 0,C 180,E1 -24651.107,E2 -24651.107} C_VEL
LIN {X 0,Y 134.893,Z 416.239,A -85,B 0,C 180,E1 -24657.014,E2 -24657.014} C_VEL
LIN {X 0,Y 134.799,Z 408.33,A -85,B 0,C 180,E1 -24662.241,E2 -24662.241} C_VEL
LIN {X 0,Y 135.157,Z 400.303,A -85,B 0,C 180,E1 -24666.634,E2 -24666.634} C_VEL
LIN {X 0,Y 135.775,Z 392.029,A -85,B 0,C 180,E1 -24670.429,E2 -24670.429} C_VEL
LIN {X 0,Y 137,Z 380.232,A -85,B 0,C 180,E1 -24674.862,E2 -24674.862} C_VEL
LIN {X 0,Y 138.445,Z 368.374,A -85,B 0,C 180,E1 -24678.498,E2 -24678.498} C_VEL
LIN {X 0,Y 140.143,Z 355.389,A -85,B 0,C 180,E1 -24681.706,E2 -24681.706} C_VEL
LIN {X 0,Y 140.27,Z 351.797,A -85,B 0,C 180,E1 -24682.46,E2 -24682.46} C_VEL
LIN {X 0,Y 137.702,Z 339.955,A -85,B 0,C 180,E1 -24684.821,E2 -24684.821} C_VEL
LIN {X 0,Y 138.445,Z 340.74,A -85,B 0,C 180,E1 -24687.084,E2 -24687.084} C_VEL
LIN {X 0,Y 140.581,Z 344.073,A -85,B 0,C 180,E1 -24689.164,E2 -24689.164} C_VEL
LIN {X 0,Y 142.959,Z 346.656,A -85,B 0,C 180,E1 -24691.18,E2 -24691.18} C_VEL
LIN {X 0,Y 145.66,Z 350.626,A -85,B 0,C 180,E1 -24693.494,E2 -24693.494} C_VEL
LIN {X 0,Y 147,Z 352.667,A -85,B 0,C 180,E1 -24694.593,E2 -24694.593} C_VEL
LIN {X 0,Y 149.803,Z 357.262,A -85,B 0,C 180,E1 -24696.918,E2 -24696.918} C_VEL
LIN {X 0,Y 153.312,Z 363.911,A -85,B 0,C 180,E1 -24699.925,E2 -24699.925} C_VEL
LIN {X 0,Y 156.693,Z 372.047,A -85,B 0,C 180,E1 -24703.158,E2 -24703.158} C_VEL
LIN {X 0,Y 158.428,Z 377.676,A -85,B 0,C 180,E1 -24705.217,E2 -24705.217} C_VEL
LIN {X 0,Y 159.332,Z 385.873,A -85,B 0,C 180,E1 -24707.803,E2 -24707.803} C_VEL
LIN {X 0,Y 159.498,Z 394.705,A -85,B 0,C 180,E1 -24710.674,E2 -24710.674} C_VEL
LIN {X 0,Y 159.08,Z 399.331,A -85,B 0,C 180,E1 -24712.195,E2 -24712.195} C_VEL
LIN {X 0,Y 155.576,Z 407.923,A -85,B 0,C 180,E1 -24714.647,E2 -24714.647} C_VEL
LIN {X 0,Y 151.528,Z 416.586,A -85,B 0,C 180,E1 -24717.766,E2 -24717.766} C_VEL
LIN {X 0,Y 147.065,Z 424.625,A -85,B 0,C 180,E1 -24721.453,E2 -24721.453} C_VEL
LIN {X 0,Y 143.414,Z 431.066,A -85,B 0,C 180,E1 -24725.383,E2 -24725.383} C_VEL
LIN {X 0,Y 140.283,Z 436.184,A -85,B 0,C 180,E1 -24729.47,E2 -24729.47} C_VEL
LIN {X 0,Y 137.82,Z 440.136,A -85,B 0,C 180,E1 -24733.712,E2 -24733.712} C_VEL
LIN {X 0,Y 136.078,Z 443.039,A -85,B 0,C 180,E1 -24738.078,E2 -24738.078} C_VEL
LIN {X 0,Y 135.227,Z 444.441,A -85,B 0,C 180,E1 -24741.03,E2 -24741.03} C_VEL
LIN {X 0,Y 134.642,Z 445.425,A -85,B 0,C 180,E1 -24744.008,E2 -24744.008} C_VEL
LIN {X 0,Y 134.144,Z 446.259,A -85,B 0,C 180,E1 -24750,E2 -24750} C_VEL
LIN {X 0,Y 134.254,Z 446.06,A -85,B 0,C 180,E1 -24753.001,E2 -24753.001} C_VEL
LIN {X 0,Y 134.62,Z 445.473,A -85,B 0,C 180,E1 -24755.993,E2 -24755.993} C_VEL
LIN {X 0,Y 135.243,Z 444.452,A -85,B 0,C 180,E1 -24759.121,E2 -24759.121} C_VEL
LIN {X 0,Y 136.026,Z 443.145,A -85,B 0,C 180,E1 -24761.927,E2 -24761.927} C_VEL
LIN {X 0,Y 137.772,Z 440.279,A -85,B 0,C 180,E1 -24766.294,E2 -24766.294} C_VEL
LIN {X 0,Y 140.23,Z 436.374,A -85,B 0,C 180,E1 -24770.538,E2 -24770.538} C_VEL
LIN {X 0,Y 143.343,Z 431.305,A -85,B 0,C 180,E1 -24774.63,E2 -24774.63} C_VEL
LIN {X 0,Y 147.012,Z 424.91,A -85,B 0,C 180,E1 -24778.559,E2 -24778.559} C_VEL
LIN {X 0,Y 151.47,Z 416.937,A -85,B 0,C 180,E1 -24782.248,E2 -24782.248} C_VEL
LIN {X 0,Y 155.395,Z 408.693,A -85,B 0,C 180,E1 -24785.259,E2 -24785.259} C_VEL
LIN {X 0,Y 159.009,Z 399.882,A -85,B 0,C 180,E1 -24787.825,E2 -24787.825} C_VEL
LIN {X 0,Y 159.409,Z 398.746,A -85,B 0,C 180,E1 -24788.114,E2 -24788.114} C_VEL
LIN {X 0,Y 159.551,Z 389.048,A -85,B 0,C 180,E1 -24791.356,E2 -24791.356} C_VEL
LIN {X 0,Y 158.814,Z 379.546,A -85,B 0,C 180,E1 -24794.353,E2 -24794.353} C_VEL
LIN {X 0,Y 157.503,Z 374.092,A -85,B 0,C 180,E1 -24796.239,E2 -24796.239} C_VEL
LIN {X 0,Y 153.954,Z 365.382,A -85,B 0,C 180,E1 -24799.71,E2 -24799.71} C_VEL
LIN {X 0,Y 150.709,Z 358.891,A -85,B 0,C 180,E1 -24802.557,E2 -24802.557} C_VEL
LIN {X 0,Y 148.545,Z 355.131,A -85,B 0,C 180,E1 -24804.371,E2 -24804.371} C_VEL
LIN {X 0,Y 146.095,Z 351.343,A -85,B 0,C 180,E1 -24806.412,E2 -24806.412} C_VEL
LIN {X 0,Y 142.395,Z 347.426,A -85,B 0,C 180,E1 -24809.404,E2 -24809.404} C_VEL
LIN {X 0,Y 141.429,Z 346.519,A -85,B 0,C 180,E1 -24810.203,E2 -24810.203} C_VEL
LIN {X 0,Y 139.619,Z 345.606,A -85,B 0,C 180,E1 -24811.676,E2 -24811.676} C_VEL
LIN {X 0,Y 137.997,Z 348.12,A -85,B 0,C 180,E1 -24812.602,E2 -24812.602} C_VEL
LIN {X 0,Y 137.019,Z 348.616,A -85,B 0,C 180,E1 -24813.333,E2 -24813.333} C_VEL
LIN {X 0,Y 136.275,Z 347.864,A -85,B 0,C 180,E1 -24814.103,E2 -24814.103} C_VEL
LIN {X 0,Y 136.099,Z 347.119,A -85,B 0,C 180,E1 -24814.375,E2 -24814.375} C_VEL
LIN {X 0,Y 138.178,Z 361.792,A -85,B 0,C 180,E1 -24816.785,E2 -24816.785} C_VEL
LIN {X 0,Y 139.617,Z 370.976,A -85,B 0,C 180,E1 -24818.595,E2 -24818.595} C_VEL
LIN {X 0,Y 138.084,Z 384.313,A -85,B 0,C 180,E1 -24821.836,E2 -24821.836} C_VEL
LIN {X 0,Y 136.577,Z 396.203,A -85,B 0,C 180,E1 -24825.471,E2 -24825.471} C_VEL
LIN {X 0,Y 135.531,Z 407.114,A -85,B 0,C 180,E1 -24829.543,E2 -24829.543} C_VEL
LIN {X 0,Y 134.773,Z 416.782,A -85,B 0,C 180,E1 -24834.013,E2 -24834.013} C_VEL
LIN {X 0,Y 134.557,Z 424.787,A -85,B 0,C 180,E1 -24838.503,E2 -24838.503} C_VEL
LIN {X 0,Y 134.654,Z 431.404,A -85,B 0,C 180,E1 -24842.992,E2 -24842.992} C_VEL
LIN {X 0,Y 135.369,Z 436.833,A -85,B 0,C 180,E1 -24847.458,E2 -24847.458} C_VEL
LIN {X 0,Y 136.794,Z 441.912,A -85,B 0,C 180,E1 -24852.536,E2 -24852.536} C_VEL
LIN {X 0,Y 139.606,Z 445.993,A -85,B 0,C 180,E1 -24857.581,E2 -24857.581} C_VEL
LIN {X 0,Y 144.132,Z 449.344,A -85,B 0,C 180,E1 -24862.96,E2 -24862.96} C_VEL
LIN {X 0,Y 150.099,Z 451.472,A -85,B 0,C 180,E1 -24867.919,E2 -24867.919} C_VEL
LIN {X 0,Y 157.264,Z 452.393,A -85,B 0,C 180,E1 -24872.43,E2 -24872.43} C_VEL
LIN {X 0,Y 165.659,Z 452.108,A -85,B 0,C 180,E1 -24876.437,E2 -24876.437} C_VEL
LIN {X 0,Y 174.99,Z 450.651,A -85,B 0,C 180,E1 -24879.986,E2 -24879.986} C_VEL
LIN {X 0,Y 185.288,Z 447.994,A -85,B 0,C 180,E1 -24883.058,E2 -24883.058} C_VEL
LIN {X 0,Y 179.12,Z 450.472,A -85,B 0,C 180,E1 -24885.069,E2 -24885.069} C_VEL
LIN {X 0,Y 169.066,Z 453.871,A -85,B 0,C 180,E1 -24888.309,E2 -24888.309} C_VEL
LIN {X 0,Y 159.963,Z 456.294,A -85,B 0,C 180,E1 -24892.041,E2 -24892.041} C_VEL
LIN {X 0,Y 152.146,Z 457.771,A -85,B 0,C 180,E1 -24896.337,E2 -24896.337} C_VEL
LIN {X 0,Y 145.642,Z 458.301,A -85,B 0,C 180,E1 -24901.148,E2 -24901.148} C_VEL
LIN {X 0,Y 140.543,Z 457.86,A -85,B 0,C 180,E1 -24906.419,E2 -24906.419} C_VEL
LIN {X 0,Y 137.101,Z 456.436,A -85,B 0,C 180,E1 -24912.087,E2 -24912.087} C_VEL
LIN {X 0,Y 136.405,Z 455.906,A -85,B 0,C 180,E1 -24913.922,E2 -24913.922} C_VEL
LIN {X 0,Y 134.917,Z 458.62,A -85,B 0,C 180,E1 -24917.973,E2 -24917.973} C_VEL
LIN {X 0,Y 134.29,Z 460.066,A -85,B 0,C 180,E1 -24920.967,E2 -24920.967} C_VEL
LIN {X 0,Y 133.894,Z 461.729,A -85,B 0,C 180,E1 -24926.991,E2 -24926.991} C_VEL
LIN {X 0,Y 134.109,Z 461.964,A -85,B 0,C 180,E1 -24930,E2 -24930} C_VEL
LIN {X 0,Y 133.857,Z 461.549,A -85,B 0,C 180,E1 -24933.993,E2 -24933.993} C_VEL
LIN {X 0,Y 133.991,Z 460.018,A -85,B 0,C 180,E1 -24939.053,E2 -24939.053} C_VEL
LIN {X 0,Y 134.498,Z 458.547,A -85,B 0,C 180,E1 -24942.065,E2 -24942.065} C_VEL
LIN {X 0,Y 135.839,Z 455.514,A -85,B 0,C 180,E1 -24946.532,E2 -24946.532} C_VEL
LIN {X 0,Y 138.193,Z 451.434,A -85,B 0,C 180,E1 -24950.855,E2 -24950.855} C_VEL
LIN {X 0,Y 140.285,Z 448.108,A -85,B 0,C 180,E1 -24953.627,E2 -24953.627} C_VEL
LIN {X 0,Y 146.493,Z 447.928,A -85,B 0,C 180,E1 -24960.282,E2 -24960.282} C_VEL
LIN {X 0,Y 155.007,Z 446.308,A -85,B 0,C 180,E1 -24966.116,E2 -24966.116} C_VEL
LIN {X 0,Y 163.269,Z 444.031,A -85,B 0,C 180,E1 -24970.217,E2 -24970.217} C_VEL
LIN {X 0,Y 170.248,Z 441.686,A -85,B 0,C 180,E1 -24972.993,E2 -24972.993} C_VEL
LIN {X 0,Y 171.266,Z 441.175,A -85,B 0,C 180,E1 -24973.753,E2 -24973.753} C_VEL
LIN {X 0,Y 171.761,Z 439.905,A -85,B 0,C 180,E1 -24976.814,E2 -24976.814} C_VEL
LIN {X 0,Y 172.794,Z 439.443,A -85,B 0,C 180,E1 -24977.409,E2 -24977.409} C_VEL
LIN {X 0,Y 174.584,Z 438.789,A -85,B 0,C 180,E1 -24978.012,E2 -24978.012} C_VEL
LIN {X 0,Y 174.014,Z 438.711,A -85,B 0,C 180,E1 -24978.761,E2 -24978.761} C_VEL
LIN {X 0,Y 167.36,Z 439.47,A -85,B 0,C 180,E1 -24980.957,E2 -24980.957} C_VEL
LIN {X 0,Y 158.01,Z 439.687,A -85,B 0,C 180,E1 -24984.675,E2 -24984.675} C_VEL
LIN {X 0,Y 149.618,Z 438.743,A -85,B 0,C 180,E1 -24988.889,E2 -24988.889} C_VEL
LIN {X 0,Y 142.517,Z 436.605,A -85,B 0,C 180,E1 -24993.652,E2 -24993.652} C_VEL
LIN {X 0,Y 136.763,Z 433.252,A -85,B 0,C 180,E1 -24998.917,E2 -24998.917} C_VEL
LIN {X 0,Y 132.421,Z 428.603,A -85,B 0,C 180,E1 -25004.611,E2 -25004.611} C_VEL
LIN {X 0,Y 129.46,Z 422.547,A -85,B 0,C 180,E1 -25010.627,E2 -25010.627} C_VEL
LIN {X 0,Y 127.922,Z 414.841,A -85,B 0,C 180,E1 -25016.851,E2 -25016.851} C_VEL
LIN {X 0,Y 127.863,Z 406.584,A -85,B 0,C 180,E1 -25022.363,E2 -25022.363} C_VEL
LIN {X 0,Y 128.223,Z 398.071,A -85,B 0,C 180,E1 -25026.996,E2 -25026.996} C_VEL
LIN {X 0,Y 129.074,Z 387.48,A -85,B 0,C 180,E1 -25031.783,E2 -25031.783} C_VEL
LIN {X 0,Y 130.255,Z 377.029,A -85,B 0,C 180,E1 -25035.651,E2 -25035.651} C_VEL
LIN {X 0,Y 131.826,Z 364.352,A -85,B 0,C 180,E1 -25039.464,E2 -25039.464} C_VEL
LIN {X 0,Y 133.192,Z 353.956,A -85,B 0,C 180,E1 -25042.016,E2 -25042.016} C_VEL
LIN {X 0,Y 132.645,Z 349.998,A -85,B 0,C 180,E1 -25042.881,E2 -25042.881} C_VEL
LIN {X 0,Y 132.529,Z 349.483,A -85,B 0,C 180,E1 -25042.988,E2 -25042.988} C_VEL
LIN {X 0,Y 133,Z 350.738,A -85,B 0,C 180,E1 -25043.76,E2 -25043.76} C_VEL
LIN {X 0,Y 134.065,Z 350.71,A -85,B 0,C 180,E1 -25044.796,E2 -25044.796} C_VEL
LIN {X 0,Y 135.669,Z 349.007,A -85,B 0,C 180,E1 -25045.918,E2 -25045.918} C_VEL
LIN {X 0,Y 136.442,Z 347.747,A -85,B 0,C 180,E1 -25046.377,E2 -25046.377} C_VEL
LIN {X 0,Y 139.554,Z 351.931,A -85,B 0,C 180,E1 -25049.615,E2 -25049.615} C_VEL
LIN {X 0,Y 143.43,Z 358.041,A -85,B 0,C 180,E1 -25053.42,E2 -25053.42} C_VEL
LIN {X 0,Y 145.509,Z 361.579,A -85,B 0,C 180,E1 -25055.422,E2 -25055.422} C_VEL
LIN {X 0,Y 149.386,Z 370.031,A -85,B 0,C 180,E1 -25059.429,E2 -25059.429} C_VEL
LIN {X 0,Y 152.291,Z 377.933,A -85,B 0,C 180,E1 -25062.809,E2 -25062.809} C_VEL
LIN {X 0,Y 153.322,Z 382.803,A -85,B 0,C 180,E1 -25064.638,E2 -25064.638} C_VEL
LIN {X 0,Y 153.734,Z 392.501,A -85,B 0,C 180,E1 -25067.945,E2 -25067.945} C_VEL
LIN {X 0,Y 153.364,Z 399.751,A -85,B 0,C 180,E1 -25070.518,E2 -25070.518} C_VEL
LIN {X 0,Y 149.66,Z 408.754,A -85,B 0,C 180,E1 -25073.214,E2 -25073.214} C_VEL
LIN {X 0,Y 145.593,Z 416.998,A -85,B 0,C 180,E1 -25076.281,E2 -25076.281} C_VEL
LIN {X 0,Y 140.886,Z 425.038,A -85,B 0,C 180,E1 -25080.076,E2 -25080.076} C_VEL
LIN {X 0,Y 137.002,Z 431.48,A -85,B 0,C 180,E1 -25084.149,E2 -25084.149} C_VEL
LIN {X 0,Y 133.672,Z 436.599,A -85,B 0,C 180,E1 -25088.405,E2 -25088.405} C_VEL
LIN {X 0,Y 131.041,Z 440.551,A -85,B 0,C 180,E1 -25092.844,E2 -25092.844} C_VEL
LIN {X 0,Y 129.157,Z 443.454,A -85,B 0,C 180,E1 -25097.428,E2 -25097.428} C_VEL
LIN {X 0,Y 128.25,Z 444.855,A -85,B 0,C 180,E1 -25100.538,E2 -25100.538} C_VEL
LIN {X 0,Y 127.608,Z 445.839,A -85,B 0,C 180,E1 -25103.676,E2 -25103.676} C_VEL
LIN {X 0,Y 127.068,Z 446.673,A -85,B 0,C 180,E1 -25110,E2 -25110} C_VEL
LIN {X 0,Y 127.19,Z 446.474,A -85,B 0,C 180,E1 -25113.168,E2 -25113.168} C_VEL
LIN {X 0,Y 128.129,Z 445.038,A -85,B 0,C 180,E1 -25119.132,E2 -25119.132} C_VEL
LIN {X 0,Y 129.103,Z 443.558,A -85,B 0,C 180,E1 -25122.577,E2 -25122.577} C_VEL
LIN {X 0,Y 130.971,Z 440.693,A -85,B 0,C 180,E1 -25127.166,E2 -25127.166} C_VEL
LIN {X 0,Y 133.623,Z 436.786,A -85,B 0,C 180,E1 -25131.603,E2 -25131.603} C_VEL
LIN {X 0,Y 136.932,Z 431.716,A -85,B 0,C 180,E1 -25135.866,E2 -25135.866} C_VEL
LIN {X 0,Y 140.836,Z 425.319,A -85,B 0,C 180,E1 -25139.935,E2 -25139.935} C_VEL
LIN {X 0,Y 145.531,Z 417.344,A -85,B 0,C 180,E1 -25143.736,E2 -25143.736} C_VEL
LIN {X 0,Y 149.943,Z 408.418,A -85,B 0,C 180,E1 -25147.062,E2 -25147.062} C_VEL
LIN {X 0,Y 153.423,Z 400.285,A -85,B 0,C 180,E1 -25149.464,E2 -25149.464} C_VEL
LIN {X 0,Y 153.787,Z 391.588,A -85,B 0,C 180,E1 -25152.574,E2 -25152.574} C_VEL
LIN {X 0,Y 153.375,Z 382.336,A -85,B 0,C 180,E1 -25155.703,E2 -25155.703} C_VEL
LIN {X 0,Y 152.142,Z 377.31,A -85,B 0,C 180,E1 -25157.655,E2 -25157.655} C_VEL
LIN {X 0,Y 148.712,Z 368.338,A -85,B 0,C 180,E1 -25161.58,E2 -25161.58} C_VEL
LIN {X 0,Y 145.096,Z 360.918,A -85,B 0,C 180,E1 -25165.226,E2 -25165.226} C_VEL
LIN {X 0,Y 142.787,Z 357.225,A -85,B 0,C 180,E1 -25167.429,E2 -25167.429} C_VEL
LIN {X 0,Y 139.427,Z 353.246,A -85,B 0,C 180,E1 -25170.563,E2 -25170.563} C_VEL
LIN {X 0,Y 137.162,Z 355.123,A -85,B 0,C 180,E1 -25171.916,E2 -25171.916} C_VEL
LIN {X 0,Y 136.239,Z 355.677,A -85,B 0,C 180,E1 -25172.545,E2 -25172.545} C_VEL
LIN {X 0,Y 134.153,Z 359.3,A -85,B 0,C 180,E1 -25173.454,E2 -25173.454} C_VEL
LIN {X 0,Y 132.423,Z 361.107,A -85,B 0,C 180,E1 -25174.498,E2 -25174.498} C_VEL
LIN {X 0,Y 131.284,Z 361.386,A -85,B 0,C 180,E1 -25175.514,E2 -25175.514} C_VEL
LIN {X 0,Y 130.764,Z 360.369,A -85,B 0,C 180,E1 -25176.384,E2 -25176.384} C_VEL
LIN {X 0,Y 130.793,Z 360.281,A -85,B 0,C 180,E1 -25176.521,E2 -25176.521} C_VEL
LIN {X 0,Y 132.467,Z 370.558,A -85,B 0,C 180,E1 -25178.607,E2 -25178.607} C_VEL
LIN {X 0,Y 131.13,Z 382.68,A -85,B 0,C 180,E1 -25181.647,E2 -25181.647} C_VEL
LIN {X 0,Y 129.608,Z 394.989,A -85,B 0,C 180,E1 -25185.475,E2 -25185.475} C_VEL
LIN {X 0,Y 128.521,Z 406.179,A -85,B 0,C 180,E1 -25189.838,E2 -25189.838} C_VEL
LIN {X 0,Y 127.8,Z 415.866,A -85,B 0,C 180,E1 -25194.477,E2 -25194.477} C_VEL
LIN {X 0,Y 127.63,Z 424.052,A -85,B 0,C 180,E1 -25199.211,E2 -25199.211} C_VEL
LIN {X 0,Y 127.913,Z 431.751,A -85,B 0,C 180,E1 -25204.727,E2 -25204.727} C_VEL
LIN {X 0,Y 128.812,Z 437.185,A -85,B 0,C 180,E1 -25209.42,E2 -25209.42} C_VEL
LIN {X 0,Y 131.018,Z 442.915,A -85,B 0,C 180,E1 -25215.558,E2 -25215.558} C_VEL
LIN {X 0,Y 135.091,Z 447.312,A -85,B 0,C 180,E1 -25221.356,E2 -25221.356} C_VEL
LIN {X 0,Y 140.511,Z 450.455,A -85,B 0,C 180,E1 -25226.754,E2 -25226.754} C_VEL
LIN {X 0,Y 147.406,Z 452.4,A -85,B 0,C 180,E1 -25231.632,E2 -25231.632} C_VEL
LIN {X 0,Y 155.573,Z 453.14,A -85,B 0,C 180,E1 -25235.964,E2 -25235.964} C_VEL
LIN {X 0,Y 164.771,Z 452.731,A -85,B 0,C 180,E1 -25239.777,E2 -25239.777} C_VEL
LIN {X 0,Y 174.923,Z 451.185,A -85,B 0,C 180,E1 -25243.08,E2 -25243.08} C_VEL
LIN {X 0,Y 174.205,Z 451.446,A -85,B 0,C 180,E1 -25243.433,E2 -25243.433} C_VEL
LIN {X 0,Y 163.842,Z 454.325,A -85,B 0,C 180,E1 -25246.66,E2 -25246.66} C_VEL
LIN {X 0,Y 154.449,Z 456.286,A -85,B 0,C 180,E1 -25250.427,E2 -25250.427} C_VEL
LIN {X 0,Y 146.316,Z 457.334,A -85,B 0,C 180,E1 -25254.802,E2 -25254.802} C_VEL
LIN {X 0,Y 139.492,Z 457.474,A -85,B 0,C 180,E1 -25259.746,E2 -25259.746} C_VEL
LIN {X 0,Y 134.133,Z 456.679,A -85,B 0,C 180,E1 -25265.218,E2 -25265.218} C_VEL
LIN {X 0,Y 130.058,Z 454.751,A -85,B 0,C 180,E1 -25272.101,E2 -25272.101} C_VEL
LIN {X 0,Y 127.962,Z 458.205,A -85,B 0,C 180,E1 -25277.309,E2 -25277.309} C_VEL
LIN {X 0,Y 127.257,Z 459.649,A -85,B 0,C 180,E1 -25280.463,E2 -25280.463} C_VEL
LIN {X 0,Y 126.828,Z 461.314,A -85,B 0,C 180,E1 -25286.823,E2 -25286.823} C_VEL
LIN {X 0,Y 127.021,Z 461.549,A -85,B 0,C 180,E1 -25290,E2 -25290} C_VEL
LIN {X 0,Y 126.773,Z 461.21,A -85,B 0,C 180,E1 -25293.732,E2 -25293.732} C_VEL
LIN {X 0,Y 126.95,Z 459.6,A -85,B 0,C 180,E1 -25299.56,E2 -25299.56} C_VEL
LIN {X 0,Y 127.542,Z 458.13,A -85,B 0,C 180,E1 -25302.733,E2 -25302.733} C_VEL
LIN {X 0,Y 128.999,Z 455.095,A -85,B 0,C 180,E1 -25307.436,E2 -25307.436} C_VEL
LIN {X 0,Y 131.562,Z 451.018,A -85,B 0,C 180,E1 -25311.959,E2 -25311.959} C_VEL
LIN {X 0,Y 134.458,Z 446.794,A -85,B 0,C 180,E1 -25315.545,E2 -25315.545} C_VEL
LIN {X 0,Y 140.291,Z 446.939,A -85,B 0,C 180,E1 -25321.61,E2 -25321.61} C_VEL
LIN {X 0,Y 149.339,Z 445.804,A -85,B 0,C 180,E1 -25327.719,E2 -25327.719} C_VEL
LIN {X 0,Y 157.92,Z 443.946,A -85,B 0,C 180,E1 -25331.879,E2 -25331.879} C_VEL
LIN {X 0,Y 167.436,Z 441.259,A -85,B 0,C 180,E1 -25335.526,E2 -25335.526} C_VEL
LIN {X 0,Y 172.794,Z 439.443,A -85,B 0,C 180,E1 -25337.409,E2 -25337.409} C_VEL
LIN {X 0,Y 173.038,Z 439.255,A -85,B 0,C 180,E1 -25337.812,E2 -25337.812} C_VEL
LIN {X 0,Y 171.867,Z 439.289,A -85,B 0,C 180,E1 -25338.509,E2 -25338.509} C_VEL
LIN {X 0,Y 168.945,Z 439.698,A -85,B 0,C 180,E1 -25339.259,E2 -25339.259} C_VEL
LIN {X 0,Y 159.787,Z 440.721,A -85,B 0,C 180,E1 -25340.662,E2 -25340.662} C_VEL
LIN {X 0,Y 156.23,Z 440.797,A -85,B 0,C 180,E1 -25341.558,E2 -25341.558} C_VEL
LIN {X 0,Y 155.617,Z 440.758,A -85,B 0,C 180,E1 -25341.783,E2 -25341.783} C_VEL
LIN {X 0,Y 147.841,Z 440.022,A -85,B 0,C 180,E1 -25345.218,E2 -25345.218} C_VEL
LIN {X 0,Y 139.708,Z 438.042,A -85,B 0,C 180,E1 -25349.798,E2 -25349.798} C_VEL
LIN {X 0,Y 133.011,Z 434.89,A -85,B 0,C 180,E1 -25354.995,E2 -25354.995} C_VEL
LIN {X 0,Y 127.735,Z 430.515,A -85,B 0,C 180,E1 -25360.724,E2 -25360.724} C_VEL
LIN {X 0,Y 123.926,Z 424.809,A -85,B 0,C 180,E1 -25366.889,E2 -25366.889} C_VEL
LIN {X 0,Y 121.367,Z 416.55,A -85,B 0,C 180,E1 -25374.184,E2 -25374.184} C_VEL
LIN {X 0,Y 120.825,Z 408.495,A -85,B 0,C 180,E1 -25380,E2 -25380} C_VEL
LIN {X 0,Y 121.099,Z 400.267,A -85,B 0,C 180,E1 -25384.994,E2 -25384.994} C_VEL
LIN {X 0,Y 121.732,Z 390.241,A -85,B 0,C 180,E1 -25389.974,E2 -25389.974} C_VEL
LIN {X 0,Y 122.861,Z 379.183,A -85,B 0,C 180,E1 -25394.493,E2 -25394.493} C_VEL
LIN {X 0,Y 124.399,Z 366.447,A -85,B 0,C 180,E1 -25398.743,E2 -25398.743} C_VEL
LIN {X 0,Y 124.783,Z 367.356,A -85,B 0,C 180,E1 -25399.751,E2 -25399.751} C_VEL
LIN {X 0,Y 126.269,Z 366.383,A -85,B 0,C 180,E1 -25401.21,E2 -25401.21} C_VEL
LIN {X 0,Y 128.949,Z 362.969,A -85,B 0,C 180,E1 -25402.99,E2 -25402.99} C_VEL
LIN {X 0,Y 131.963,Z 357.967,A -85,B 0,C 180,E1 -25404.525,E2 -25404.525} C_VEL
LIN {X 0,Y 134.297,Z 356.827,A -85,B 0,C 180,E1 -25406.412,E2 -25406.412} C_VEL
LIN {X 0,Y 135.212,Z 356.182,A -85,B 0,C 180,E1 -25407.053,E2 -25407.053} C_VEL
LIN {X 0,Y 137.318,Z 359.165,A -85,B 0,C 180,E1 -25409.452,E2 -25409.452} C_VEL
LIN {X 0,Y 140.075,Z 364.07,A -85,B 0,C 180,E1 -25412.64,E2 -25412.64} C_VEL
LIN {X 0,Y 141.651,Z 366.979,A -85,B 0,C 180,E1 -25414.421,E2 -25414.421} C_VEL
LIN {X 0,Y 144.739,Z 374.475,A -85,B 0,C 180,E1 -25418.25,E2 -25418.25} C_VEL
LIN {X 0,Y 147.283,Z 382.403,A -85,B 0,C 180,E1 -25421.917,E2 -25421.917} C_VEL
LIN {X 0,Y 147.935,Z 386.479,A -85,B 0,C 180,E1 -25423.563,E2 -25423.563} C_VEL
LIN {X 0,Y 147.967,Z 395.105,A -85,B 0,C 180,E1 -25426.729,E2 -25426.729} C_VEL
LIN {X 0,Y 147.48,Z 401.259,A -85,B 0,C 180,E1 -25429.062,E2 -25429.062} C_VEL
LIN {X 0,Y 144.852,Z 407.291,A -85,B 0,C 180,E1 -25430.895,E2 -25430.895} C_VEL
LIN {X 0,Y 141.498,Z 414.284,A -85,B 0,C 180,E1 -25433.414,E2 -25433.414} C_VEL
LIN {X 0,Y 136.363,Z 422.977,A -85,B 0,C 180,E1 -25437.237,E2 -25437.237} C_VEL
LIN {X 0,Y 132.051,Z 429.919,A -85,B 0,C 180,E1 -25441.38,E2 -25441.38} C_VEL
LIN {X 0,Y 128.207,Z 435.437,A -85,B 0,C 180,E1 -25445.724,E2 -25445.724} C_VEL
LIN {X 0,Y 125.134,Z 439.757,A -85,B 0,C 180,E1 -25450.307,E2 -25450.307} C_VEL
LIN {X 0,Y 123.503,Z 442.026,A -85,B 0,C 180,E1 -25453.469,E2 -25453.469} C_VEL
LIN {X 0,Y 122.253,Z 443.869,A -85,B 0,C 180,E1 -25456.706,E2 -25456.706} C_VEL
LIN {X 0,Y 121.185,Z 445.395,A -85,B 0,C 180,E1 -25460.37,E2 -25460.37} C_VEL
LIN {X 0,Y 120.133,Z 446.86,A -85,B 0,C 180,E1 -25466.646,E2 -25466.646} C_VEL
LIN {X 0,Y 119.994,Z 447.087,A -85,B 0,C 180,E1 -25470,E2 -25470} C_VEL
LIN {X 0,Y 120.128,Z 446.888,A -85,B 0,C 180,E1 -25473.354,E2 -25473.354} C_VEL
LIN {X 0,Y 121.236,Z 445.335,A -85,B 0,C 180,E1 -25480.015,E2 -25480.015} C_VEL
LIN {X 0,Y 122.185,Z 443.973,A -85,B 0,C 180,E1 -25483.302,E2 -25483.302} C_VEL
LIN {X 0,Y 124.212,Z 441.106,A -85,B 0,C 180,E1 -25488.131,E2 -25488.131} C_VEL
LIN {X 0,Y 127.071,Z 437.197,A -85,B 0,C 180,E1 -25492.778,E2 -25492.778} C_VEL
LIN {X 0,Y 130.595,Z 432.127,A -85,B 0,C 180,E1 -25497.222,E2 -25497.222} C_VEL
LIN {X 0,Y 134.75,Z 425.728,A -85,B 0,C 180,E1 -25501.437,E2 -25501.437} C_VEL
LIN {X 0,Y 139.702,Z 417.751,A -85,B 0,C 180,E1 -25505.348,E2 -25505.348} C_VEL
LIN {X 0,Y 143.695,Z 410.168,A -85,B 0,C 180,E1 -25508.288,E2 -25508.288} C_VEL
LIN {X 0,Y 147.512,Z 401.747,A -85,B 0,C 180,E1 -25510.927,E2 -25510.927} C_VEL
LIN {X 0,Y 148.036,Z 394.382,A -85,B 0,C 180,E1 -25513.746,E2 -25513.746} C_VEL
LIN {X 0,Y 148.012,Z 385.973,A -85,B 0,C 180,E1 -25516.803,E2 -25516.803} C_VEL
LIN {X 0,Y 146.963,Z 381.057,A -85,B 0,C 180,E1 -25518.888,E2 -25518.888} C_VEL
LIN {X 0,Y 144.379,Z 373.401,A -85,B 0,C 180,E1 -25522.521,E2 -25522.521} C_VEL
LIN {X 0,Y 141.5,Z 366.704,A -85,B 0,C 180,E1 -25526.026,E2 -25526.026} C_VEL
LIN {X 0,Y 139.139,Z 362.81,A -85,B 0,C 180,E1 -25528.608,E2 -25528.608} C_VEL
LIN {X 0,Y 137.629,Z 361.064,A -85,B 0,C 180,E1 -25530.14,E2 -25530.14} C_VEL
LIN {X 0,Y 136.844,Z 361.643,A -85,B 0,C 180,E1 -25530.586,E2 -25530.586} C_VEL
LIN {X 0,Y 135.173,Z 364.05,A -85,B 0,C 180,E1 -25531.253,E2 -25531.253} C_VEL
LIN {X 0,Y 133.948,Z 365.45,A -85,B 0,C 180,E1 -25531.822,E2 -25531.822} C_VEL
LIN {X 0,Y 131.638,Z 367.423,A -85,B 0,C 180,E1 -25533.157,E2 -25533.157} C_VEL
LIN {X 0,Y 130.056,Z 368.103,A -85,B 0,C 180,E1 -25534.386,E2 -25534.386} C_VEL
LIN {X 0,Y 129.04,Z 368.964,A -85,B 0,C 180,E1 -25535.059,E2 -25535.059} C_VEL
LIN {X 0,Y 127.367,Z 370.796,A -85,B 0,C 180,E1 -25536.043,E2 -25536.043} C_VEL
LIN {X 0,Y 126.154,Z 371.503,A -85,B 0,C 180,E1 -25537.047,E2 -25537.047} C_VEL
LIN {X 0,Y 125.261,Z 370.367,A -85,B 0,C 180,E1 -25538.665,E2 -25538.665} C_VEL
LIN {X 0,Y 124.175,Z 381.017,A -85,B 0,C 180,E1 -25541.436,E2 -25541.436} C_VEL
LIN {X 0,Y 122.816,Z 392.329,A -85,B 0,C 180,E1 -25545.078,E2 -25545.078} C_VEL
LIN {X 0,Y 121.75,Z 403.079,A -85,B 0,C 180,E1 -25549.266,E2 -25549.266} C_VEL
LIN {X 0,Y 120.93,Z 413.336,A -85,B 0,C 180,E1 -25554.163,E2 -25554.163} C_VEL
LIN {X 0,Y 120.736,Z 421.865,A -85,B 0,C 180,E1 -25559.166,E2 -25559.166} C_VEL
LIN {X 0,Y 121.026,Z 430.025,A -85,B 0,C 180,E1 -25564.997,E2 -25564.997} C_VEL
LIN {X 0,Y 121.958,Z 435.717,A -85,B 0,C 180,E1 -25569.955,E2 -25569.955} C_VEL
LIN {X 0,Y 124.288,Z 441.86,A -85,B 0,C 180,E1 -25576.423,E2 -25576.423} C_VEL
LIN {X 0,Y 128.548,Z 446.655,A -85,B 0,C 180,E1 -25582.501,E2 -25582.501} C_VEL
LIN {X 0,Y 134.224,Z 450.174,A -85,B 0,C 180,E1 -25588.115,E2 -25588.115} C_VEL
LIN {X 0,Y 141.418,Z 452.512,A -85,B 0,C 180,E1 -25593.138,E2 -25593.138} C_VEL
LIN {X 0,Y 149.918,Z 453.702,A -85,B 0,C 180,E1 -25597.548,E2 -25597.548} C_VEL
LIN {X 0,Y 159.433,Z 453.768,A -85,B 0,C 180,E1 -25601.393,E2 -25601.393} C_VEL
LIN {X 0,Y 164.05,Z 453.503,A -85,B 0,C 180,E1 -25603.257,E2 -25603.257} C_VEL
LIN {X 0,Y 153.802,Z 455.446,A -85,B 0,C 180,E1 -25606.731,E2 -25606.731} C_VEL
LIN {X 0,Y 144.65,Z 456.506,A -85,B 0,C 180,E1 -25610.83,E2 -25610.83} C_VEL
LIN {X 0,Y 136.872,Z 456.699,A -85,B 0,C 180,E1 -25615.61,E2 -25615.61} C_VEL
LIN {X 0,Y 130.445,Z 456.015,A -85,B 0,C 180,E1 -25620.994,E2 -25620.994} C_VEL
LIN {X 0,Y 125.654,Z 454.409,A -85,B 0,C 180,E1 -25626.951,E2 -25626.951} C_VEL
LIN {X 0,Y 124.051,Z 453.398,A -85,B 0,C 180,E1 -25629.912,E2 -25629.912} C_VEL
LIN {X 0,Y 122.239,Z 455.882,A -85,B 0,C 180,E1 -25633.293,E2 -25633.293} C_VEL
LIN {X 0,Y 121.038,Z 457.79,A -85,B 0,C 180,E1 -25636.57,E2 -25636.57} C_VEL
LIN {X 0,Y 120.245,Z 459.233,A -85,B 0,C 180,E1 -25639.901,E2 -25639.901} C_VEL
LIN {X 0,Y 119.751,Z 460.9,A -85,B 0,C 180,E1 -25646.635,E2 -25646.635} C_VEL
LIN {X 0,Y 119.935,Z 461.134,A -85,B 0,C 180,E1 -25650,E2 -25650} C_VEL
LIN {X 0,Y 119.683,Z 460.882,A -85,B 0,C 180,E1 -25653.366,E2 -25653.366} C_VEL
LIN {X 0,Y 119.672,Z 460.23,A -85,B 0,C 180,E1 -25656.745,E2 -25656.745} C_VEL
LIN {X 0,Y 119.938,Z 459.183,A -85,B 0,C 180,E1 -25660.125,E2 -25660.125} C_VEL
LIN {X 0,Y 120.583,Z 457.712,A -85,B 0,C 180,E1 -25663.482,E2 -25663.482} C_VEL
LIN {X 0,Y 122.206,Z 454.677,A -85,B 0,C 180,E1 -25668.44,E2 -25668.44} C_VEL
LIN {X 0,Y 124.991,Z 450.601,A -85,B 0,C 180,E1 -25673.178,E2 -25673.178} C_VEL
LIN {X 0,Y 128.787,Z 445.362,A -85,B 0,C 180,E1 -25677.636,E2 -25677.636} C_VEL
LIN {X 0,Y 136.167,Z 445.752,A -85,B 0,C 180,E1 -25684.593,E2 -25684.593} C_VEL
LIN {X 0,Y 143.819,Z 445.121,A -85,B 0,C 180,E1 -25689.44,E2 -25689.44} C_VEL
LIN {X 0,Y 152.717,Z 443.676,A -85,B 0,C 180,E1 -25693.654,E2 -25693.654} C_VEL
LIN {X 0,Y 162.545,Z 441.437,A -85,B 0,C 180,E1 -25697.31,E2 -25697.31} C_VEL
LIN {X 0,Y 163.863,Z 441.061,A -85,B 0,C 180,E1 -25697.779,E2 -25697.779} C_VEL
LIN {X 0,Y 164.581,Z 440.694,A -85,B 0,C 180,E1 -25698.542,E2 -25698.542} C_VEL
LIN {X 0,Y 155.617,Z 440.758,A -85,B 0,C 180,E1 -25701.783,E2 -25701.783} C_VEL
LIN {X 0,Y 151.203,Z 440.599,A -85,B 0,C 180,E1 -25703.248,E2 -25703.248} C_VEL
LIN {X 0,Y 142.977,Z 439.902,A -85,B 0,C 180,E1 -25705.388,E2 -25705.388} C_VEL
LIN {X 0,Y 135.183,Z 438.458,A -85,B 0,C 180,E1 -25707.81,E2 -25707.81} C_VEL
LIN {X 0,Y 131.55,Z 437.17,A -85,B 0,C 180,E1 -25709.723,E2 -25709.723} C_VEL
LIN {X 0,Y 125.113,Z 433.464,A -85,B 0,C 180,E1 -25715.083,E2 -25715.083} C_VEL
LIN {X 0,Y 119.961,Z 428.367,A -85,B 0,C 180,E1 -25721.203,E2 -25721.203} C_VEL
LIN {X 0,Y 116.337,Z 421.897,A -85,B 0,C 180,E1 -25727.794,E2 -25727.794} C_VEL
LIN {X 0,Y 114.31,Z 413.8,A -85,B 0,C 180,E1 -25734.709,E2 -25734.709} C_VEL
LIN {X 0,Y 113.958,Z 405.153,A -85,B 0,C 180,E1 -25740.884,E2 -25740.884} C_VEL
LIN {X 0,Y 114.215,Z 397.792,A -85,B 0,C 180,E1 -25745.296,E2 -25745.296} C_VEL
LIN {X 0,Y 114.868,Z 387.295,A -85,B 0,C 180,E1 -25750.577,E2 -25750.577} C_VEL
LIN {X 0,Y 115.563,Z 380.788,A -85,B 0,C 180,E1 -25753.452,E2 -25753.452} C_VEL
LIN {X 0,Y 115.595,Z 381.322,A -85,B 0,C 180,E1 -25754.075,E2 -25754.075} C_VEL
LIN {X 0,Y 117.397,Z 380.282,A -85,B 0,C 180,E1 -25756.695,E2 -25756.695} C_VEL
LIN {X 0,Y 120.037,Z 377.371,A -85,B 0,C 180,E1 -25758.785,E2 -25758.785} C_VEL
LIN {X 0,Y 122.333,Z 374.331,A -85,B 0,C 180,E1 -25760.164,E2 -25760.164} C_VEL
LIN {X 0,Y 125.586,Z 372.159,A -85,B 0,C 180,E1 -25763.063,E2 -25763.063} C_VEL
LIN {X 0,Y 127.871,Z 369.749,A -85,B 0,C 180,E1 -25764.453,E2 -25764.453} C_VEL
LIN {X 0,Y 131.421,Z 365.069,A -85,B 0,C 180,E1 -25766.18,E2 -25766.18} C_VEL
LIN {X 0,Y 132.482,Z 363.993,A -85,B 0,C 180,E1 -25766.803,E2 -25766.803} C_VEL
LIN {X 0,Y 133.882,Z 364.604,A -85,B 0,C 180,E1 -25768.193,E2 -25768.193} C_VEL
LIN {X 0,Y 137.005,Z 371.088,A -85,B 0,C 180,E1 -25772.59,E2 -25772.59} C_VEL
LIN {X 0,Y 139.569,Z 377.542,A -85,B 0,C 180,E1 -25776.324,E2 -25776.324} C_VEL
LIN {X 0,Y 141.753,Z 384.994,A -85,B 0,C 180,E1 -25780.131,E2 -25780.131} C_VEL
LIN {X 0,Y 142.524,Z 389.753,A -85,B 0,C 180,E1 -25782.297,E2 -25782.297} C_VEL
LIN {X 0,Y 142.212,Z 398.132,A -85,B 0,C 180,E1 -25785.609,E2 -25785.609} C_VEL
LIN {X 0,Y 141.363,Z 403.742,A -85,B 0,C 180,E1 -25787.843,E2 -25787.843} C_VEL
LIN {X 0,Y 137.142,Z 412.394,A -85,B 0,C 180,E1 -25790.747,E2 -25790.747} C_VEL
LIN {X 0,Y 132.195,Z 420.729,A -85,B 0,C 180,E1 -25794.211,E2 -25794.211} C_VEL
LIN {X 0,Y 127.292,Z 428.173,A -85,B 0,C 180,E1 -25798.365,E2 -25798.365} C_VEL
LIN {X 0,Y 123.063,Z 434.138,A -85,B 0,C 180,E1 -25802.814,E2 -25802.814} C_VEL
LIN {X 0,Y 119.513,Z 438.847,A -85,B 0,C 180,E1 -25807.528,E2 -25807.528} C_VEL
LIN {X 0,Y 116.717,Z 442.441,A -85,B 0,C 180,E1 -25812.478,E2 -25812.478} C_VEL
LIN {X 0,Y 115.357,Z 444.285,A -85,B 0,C 180,E1 -25815.895,E2 -25815.895} C_VEL
LIN {X 0,Y 114.068,Z 445.984,A -85,B 0,C 180,E1 -25820.334,E2 -25820.334} C_VEL
LIN {X 0,Y 113.074,Z 447.274,A -85,B 0,C 180,E1 -25826.437,E2 -25826.437} C_VEL
LIN {X 0,Y 112.922,Z 447.501,A -85,B 0,C 180,E1 -25830,E2 -25830} C_VEL
LIN {X 0,Y 113.069,Z 447.302,A -85,B 0,C 180,E1 -25833.564,E2 -25833.564} C_VEL
LIN {X 0,Y 114.26,Z 445.75,A -85,B 0,C 180,E1 -25840.634,E2 -25840.634} C_VEL
LIN {X 0,Y 115.309,Z 444.386,A -85,B 0,C 180,E1 -25844.111,E2 -25844.111} C_VEL
LIN {X 0,Y 117.504,Z 441.519,A -85,B 0,C 180,E1 -25849.206,E2 -25849.206} C_VEL
LIN {X 0,Y 120.565,Z 437.61,A -85,B 0,C 180,E1 -25854.082,E2 -25854.082} C_VEL
LIN {X 0,Y 124.339,Z 432.538,A -85,B 0,C 180,E1 -25858.715,E2 -25858.715} C_VEL
LIN {X 0,Y 128.767,Z 426.137,A -85,B 0,C 180,E1 -25863.079,E2 -25863.079} C_VEL
LIN {X 0,Y 133.981,Z 418.159,A -85,B 0,C 180,E1 -25867.102,E2 -25867.102} C_VEL
LIN {X 0,Y 139.01,Z 408.965,A -85,B 0,C 180,E1 -25870.68,E2 -25870.68} C_VEL
LIN {X 0,Y 141.681,Z 403.197,A -85,B 0,C 180,E1 -25872.521,E2 -25872.521} C_VEL
LIN {X 0,Y 142.491,Z 394.808,A -85,B 0,C 180,E1 -25875.925,E2 -25875.925} C_VEL
LIN {X 0,Y 142.58,Z 388.835,A -85,B 0,C 180,E1 -25878.282,E2 -25878.282} C_VEL
LIN {X 0,Y 141.082,Z 382.19,A -85,B 0,C 180,E1 -25881.487,E2 -25881.487} C_VEL
LIN {X 0,Y 138.744,Z 375.141,A -85,B 0,C 180,E1 -25885.258,E2 -25885.258} C_VEL
LIN {X 0,Y 136.151,Z 369.252,A -85,B 0,C 180,E1 -25888.923,E2 -25888.923} C_VEL
LIN {X 0,Y 131.486,Z 372.989,A -85,B 0,C 180,E1 -25891.245,E2 -25891.245} C_VEL
LIN {X 0,Y 129.488,Z 374.143,A -85,B 0,C 180,E1 -25892.526,E2 -25892.526} C_VEL
LIN {X 0,Y 125.283,Z 377.349,A -85,B 0,C 180,E1 -25895.119,E2 -25895.119} C_VEL
LIN {X 0,Y 123.632,Z 378.051,A -85,B 0,C 180,E1 -25896.551,E2 -25896.551} C_VEL
LIN {X 0,Y 122.694,Z 378.794,A -85,B 0,C 180,E1 -25897.224,E2 -25897.224} C_VEL
LIN {X 0,Y 120.195,Z 381.712,A -85,B 0,C 180,E1 -25898.534,E2 -25898.534} C_VEL
LIN {X 0,Y 119.084,Z 382.775,A -85,B 0,C 180,E1 -25899.261,E2 -25899.261} C_VEL
LIN {X 0,Y 116.809,Z 383.101,A -85,B 0,C 180,E1 -25902.492,E2 -25902.492} C_VEL
LIN {X 0,Y 115.323,Z 395.451,A -85,B 0,C 180,E1 -25906.878,E2 -25906.878} C_VEL
LIN {X 0,Y 114.526,Z 404.453,A -85,B 0,C 180,E1 -25910.773,E2 -25910.773} C_VEL
LIN {X 0,Y 113.927,Z 415.195,A -85,B 0,C 180,E1 -25916.463,E2 -25916.463} C_VEL
LIN {X 0,Y 113.907,Z 423.45,A -85,B 0,C 180,E1 -25921.768,E2 -25921.768} C_VEL
LIN {X 0,Y 114.436,Z 430.194,A -85,B 0,C 180,E1 -25927.055,E2 -25927.055} C_VEL
LIN {X 0,Y 115.749,Z 436.417,A -85,B 0,C 180,E1 -25932.819,E2 -25932.819} C_VEL
LIN {X 0,Y 118.595,Z 442.027,A -85,B 0,C 180,E1 -25939.022,E2 -25939.022} C_VEL
LIN {X 0,Y 123.434,Z 446.864,A -85,B 0,C 180,E1 -25945.279,E2 -25945.279} C_VEL
LIN {X 0,Y 128.028,Z 449.701,A -85,B 0,C 180,E1 -25949.607,E2 -25949.607} C_VEL
LIN {X 0,Y 135.545,Z 452.441,A -85,B 0,C 180,E1 -25954.775,E2 -25954.775} C_VEL
LIN {X 0,Y 144.373,Z 454.082,A -85,B 0,C 180,E1 -25959.259,E2 -25959.259} C_VEL
LIN {X 0,Y 153.838,Z 454.632,A -85,B 0,C 180,E1 -25963.034,E2 -25963.034} C_VEL
LIN {X 0,Y 143.803,Z 455.676,A -85,B 0,C 180,E1 -25966.826,E2 -25966.826} C_VEL
LIN {X 0,Y 135.019,Z 455.889,A -85,B 0,C 180,E1 -25971.345,E2 -25971.345} C_VEL
LIN {X 0,Y 127.579,Z 455.27,A -85,B 0,C 180,E1 -25976.573,E2 -25976.573} C_VEL
LIN {X 0,Y 121.626,Z 453.777,A -85,B 0,C 180,E1 -25982.466,E2 -25982.466} C_VEL
LIN {X 0,Y 118.263,Z 451.975,A -85,B 0,C 180,E1 -25987.508,E2 -25987.508} C_VEL
LIN {X 0,Y 115.447,Z 455.468,A -85,B 0,C 180,E1 -25992.279,E2 -25992.279} C_VEL
LIN {X 0,Y 114.146,Z 457.375,A -85,B 0,C 180,E1 -25995.742,E2 -25995.742} C_VEL
LIN {X 0,Y 113.263,Z 458.818,A -85,B 0,C 180,E1 -25999.272,E2 -25999.272} C_VEL
LIN {X 0,Y 112.668,Z 460.484,A -85,B 0,C 180,E1 -26006.424,E2 -26006.424} C_VEL
LIN {X 0,Y 112.85,Z 460.719,A -85,B 0,C 180,E1 -26010,E2 -26010} C_VEL
LIN {X 0,Y 112.586,Z 460.465,A -85,B 0,C 180,E1 -26013.579,E2 -26013.579} C_VEL
LIN {X 0,Y 112.598,Z 459.813,A -85,B 0,C 180,E1 -26017.171,E2 -26017.171} C_VEL
LIN {X 0,Y 112.923,Z 458.765,A -85,B 0,C 180,E1 -26020.761,E2 -26020.761} C_VEL
LIN {X 0,Y 113.656,Z 457.293,A -85,B 0,C 180,E1 -26024.32,E2 -26024.32} C_VEL
LIN {X 0,Y 115.465,Z 454.259,A -85,B 0,C 180,E1 -26029.559,E2 -26029.559} C_VEL
LIN {X 0,Y 118.49,Z 450.185,A -85,B 0,C 180,E1 -26034.532,E2 -26034.532} C_VEL
LIN {X 0,Y 122.517,Z 444.943,A -85,B 0,C 180,E1 -26039.182,E2 -26039.182} C_VEL
LIN {X 0,Y 123.515,Z 443.887,A -85,B 0,C 180,E1 -26040.095,E2 -26040.095} C_VEL
LIN {X 0,Y 130.455,Z 444.51,A -85,B 0,C 180,E1 -26046.342,E2 -26046.342} C_VEL
LIN {X 0,Y 138.443,Z 444.243,A -85,B 0,C 180,E1 -26051.295,E2 -26051.295} C_VEL
LIN {X 0,Y 147.676,Z 443.204,A -85,B 0,C 180,E1 -26055.55,E2 -26055.55} C_VEL
LIN {X 0,Y 153.89,Z 442.185,A -85,B 0,C 180,E1 -26057.815,E2 -26057.815} C_VEL
LIN {X 0,Y 154.325,Z 441.907,A -85,B 0,C 180,E1 -26058.568,E2 -26058.568} C_VEL
LIN {X 0,Y 146.721,Z 441.29,A -85,B 0,C 180,E1 -26061.486,E2 -26061.486} C_VEL
LIN {X 0,Y 137.67,Z 439.439,A -85,B 0,C 180,E1 -26065.837,E2 -26065.837} C_VEL
LIN {X 0,Y 131.55,Z 437.17,A -85,B 0,C 180,E1 -26069.723,E2 -26069.723} C_VEL
LIN {X 0,Y 128.135,Z 435.75,A -85,B 0,C 180,E1 -26071.751,E2 -26071.751} C_VEL
LIN {X 0,Y 121.485,Z 432.783,A -85,B 0,C 180,E1 -26074.849,E2 -26074.849} C_VEL
LIN {X 0,Y 115.387,Z 429.209,A -85,B 0,C 180,E1 -26078.218,E2 -26078.218} C_VEL
LIN {X 0,Y 112.948,Z 426.798,A -85,B 0,C 180,E1 -26080.633,E2 -26080.633} C_VEL
LIN {X 0,Y 109.556,Z 420.428,A -85,B 0,C 180,E1 -26087.025,E2 -26087.025} C_VEL
LIN {X 0,Y 107.585,Z 413.057,A -85,B 0,C 180,E1 -26093.436,E2 -26093.436} C_VEL
LIN {X 0,Y 107.094,Z 404.257,A -85,B 0,C 180,E1 -26100,E2 -26100} C_VEL
LIN {X 0,Y 107.295,Z 396.755,A -85,B 0,C 180,E1 -26104.697,E2 -26104.697} C_VEL
LIN {X 0,Y 107.443,Z 392.518,A -85,B 0,C 180,E1 -26107.045,E2 -26107.045} C_VEL
LIN {X 0,Y 107.334,Z 392.841,A -85,B 0,C 180,E1 -26107.525,E2 -26107.525} C_VEL
LIN {X 0,Y 108.833,Z 391.825,A -85,B 0,C 180,E1 -26111.171,E2 -26111.171} C_VEL
LIN {X 0,Y 109.822,Z 390.813,A -85,B 0,C 180,E1 -26112.392,E2 -26112.392} C_VEL
LIN {X 0,Y 112.225,Z 388.114,A -85,B 0,C 180,E1 -26114.507,E2 -26114.507} C_VEL
LIN {X 0,Y 114.847,Z 386.472,A -85,B 0,C 180,E1 -26117.817,E2 -26117.817} C_VEL
LIN {X 0,Y 116.544,Z 385.085,A -85,B 0,C 180,E1 -26119.37,E2 -26119.37} C_VEL
LIN {X 0,Y 119.989,Z 381.544,A -85,B 0,C 180,E1 -26121.564,E2 -26121.564} C_VEL
LIN {X 0,Y 121.33,Z 380.015,A -85,B 0,C 180,E1 -26122.297,E2 -26122.297} C_VEL
LIN {X 0,Y 124.767,Z 377.814,A -85,B 0,C 180,E1 -26124.991,E2 -26124.991} C_VEL
LIN {X 0,Y 128.315,Z 374.371,A -85,B 0,C 180,E1 -26126.864,E2 -26126.864} C_VEL
LIN {X 0,Y 130.858,Z 371.578,A -85,B 0,C 180,E1 -26128.03,E2 -26128.03} C_VEL
LIN {X 0,Y 133.15,Z 376.818,A -85,B 0,C 180,E1 -26131.859,E2 -26131.859} C_VEL
LIN {X 0,Y 135.219,Z 383.099,A -85,B 0,C 180,E1 -26135.707,E2 -26135.707} C_VEL
LIN {X 0,Y 136.947,Z 390.789,A -85,B 0,C 180,E1 -26139.901,E2 -26139.901} C_VEL
LIN {X 0,Y 137.036,Z 395.021,A -85,B 0,C 180,E1 -26141.814,E2 -26141.814} C_VEL
LIN {X 0,Y 136.125,Z 403.155,A -85,B 0,C 180,E1 -26145.296,E2 -26145.296} C_VEL
LIN {X 0,Y 135.691,Z 405.194,A -85,B 0,C 180,E1 -26146.152,E2 -26146.152} C_VEL
LIN {X 0,Y 131.015,Z 414.075,A -85,B 0,C 180,E1 -26149.278,E2 -26149.278} C_VEL
LIN {X 0,Y 125.611,Z 422.475,A -85,B 0,C 180,E1 -26153.025,E2 -26153.025} C_VEL
LIN {X 0,Y 120.539,Z 429.677,A -85,B 0,C 180,E1 -26157.363,E2 -26157.363} C_VEL
LIN {X 0,Y 115.436,Z 436.267,A -85,B 0,C 180,E1 -26162.831,E2 -26162.831} C_VEL
LIN {X 0,Y 111.89,Z 440.587,A -85,B 0,C 180,E1 -26167.86,E2 -26167.86} C_VEL
LIN {X 0,Y 109.983,Z 442.856,A -85,B 0,C 180,E1 -26171.367,E2 -26171.367} C_VEL
LIN {X 0,Y 108.507,Z 444.7,A -85,B 0,C 180,E1 -26174.984,E2 -26174.984} C_VEL
LIN {X 0,Y 106.933,Z 446.591,A -85,B 0,C 180,E1 -26180.352,E2 -26180.352} C_VEL
LIN {X 0,Y 106.018,Z 447.689,A -85,B 0,C 180,E1 -26186.199,E2 -26186.199} C_VEL
LIN {X 0,Y 105.852,Z 447.915,A -85,B 0,C 180,E1 -26190,E2 -26190} C_VEL
LIN {X 0,Y 106.012,Z 447.716,A -85,B 0,C 180,E1 -26193.801,E2 -26193.801} C_VEL
LIN {X 0,Y 107.307,Z 446.164,A -85,B 0,C 180,E1 -26201.331,E2 -26201.331} C_VEL
LIN {X 0,Y 108.448,Z 444.8,A -85,B 0,C 180,E1 -26205.024,E2 -26205.024} C_VEL
LIN {X 0,Y 110.848,Z 441.932,A -85,B 0,C 180,E1 -26210.409,E2 -26210.409} C_VEL
LIN {X 0,Y 114.12,Z 438.023,A -85,B 0,C 180,E1 -26215.537,E2 -26215.537} C_VEL
LIN {X 0,Y 118.178,Z 432.948,A -85,B 0,C 180,E1 -26220.364,E2 -26220.364} C_VEL
LIN {X 0,Y 122.894,Z 426.546,A -85,B 0,C 180,E1 -26224.881,E2 -26224.881} C_VEL
LIN {X 0,Y 128.391,Z 418.566,A -85,B 0,C 180,E1 -26229.013,E2 -26229.013} C_VEL
LIN {X 0,Y 133.461,Z 409.841,A -85,B 0,C 180,E1 -26232.503,E2 -26232.503} C_VEL
LIN {X 0,Y 135.993,Z 404.646,A -85,B 0,C 180,E1 -26234.241,E2 -26234.241} C_VEL
LIN {X 0,Y 137.009,Z 396.757,A -85,B 0,C 180,E1 -26237.668,E2 -26237.668} C_VEL
LIN {X 0,Y 137.157,Z 391.836,A -85,B 0,C 180,E1 -26239.801,E2 -26239.801} C_VEL
LIN {X 0,Y 136.272,Z 386.973,A -85,B 0,C 180,E1 -26242.355,E2 -26242.355} C_VEL
LIN {X 0,Y 134.497,Z 380.519,A -85,B 0,C 180,E1 -26246.074,E2 -26246.074} C_VEL
LIN {X 0,Y 133.333,Z 377.167,A -85,B 0,C 180,E1 -26248.19,E2 -26248.19} C_VEL
LIN {X 0,Y 126.567,Z 381.394,A -85,B 0,C 180,E1 -26251.836,E2 -26251.836} C_VEL
LIN {X 0,Y 124.352,Z 382.896,A -85,B 0,C 180,E1 -26253.119,E2 -26253.119} C_VEL
LIN {X 0,Y 122.44,Z 383.88,A -85,B 0,C 180,E1 -26254.501,E2 -26254.501} C_VEL
LIN {X 0,Y 121.362,Z 384.692,A -85,B 0,C 180,E1 -26255.175,E2 -26255.175} C_VEL
LIN {X 0,Y 117.702,Z 388.118,A -85,B 0,C 180,E1 -26257.1,E2 -26257.1} C_VEL
LIN {X 0,Y 115.958,Z 389.035,A -85,B 0,C 180,E1 -26258.675,E2 -26258.675} C_VEL
LIN {X 0,Y 114.741,Z 389.204,A -85,B 0,C 180,E1 -26260.313,E2 -26260.313} C_VEL
LIN {X 0,Y 112.343,Z 391.712,A -85,B 0,C 180,E1 -26261.772,E2 -26261.772} C_VEL
LIN {X 0,Y 109.667,Z 394.041,A -85,B 0,C 180,E1 -26264.004,E2 -26264.004} C_VEL
LIN {X 0,Y 108.875,Z 394.538,A -85,B 0,C 180,E1 -26265.036,E2 -26265.036} C_VEL
LIN {X 0,Y 108.357,Z 394.14,A -85,B 0,C 180,E1 -26266.962,E2 -26266.962} C_VEL
LIN {X 0,Y 108.37,Z 394.365,A -85,B 0,C 180,E1 -26267.269,E2 -26267.269} C_VEL
LIN {X 0,Y 107.552,Z 403.965,A -85,B 0,C 180,E1 -26271.665,E2 -26271.665} C_VEL
LIN {X 0,Y 107.067,Z 413.952,A -85,B 0,C 180,E1 -26277.178,E2 -26277.178} C_VEL
LIN {X 0,Y 107.16,Z 422.266,A -85,B 0,C 180,E1 -26282.819,E2 -26282.819} C_VEL
LIN {X 0,Y 108.019,Z 430.315,A -85,B 0,C 180,E1 -26289.361,E2 -26289.361} C_VEL
LIN {X 0,Y 110.156,Z 437.561,A -85,B 0,C 180,E1 -26296.685,E2 -26296.685} C_VEL
LIN {X 0,Y 114.375,Z 443.456,A -85,B 0,C 180,E1 -26303.541,E2 -26303.541} C_VEL
LIN {X 0,Y 118.638,Z 447.039,A -85,B 0,C 180,E1 -26308.288,E2 -26308.288} C_VEL
LIN {X 0,Y 125.751,Z 450.742,A -85,B 0,C 180,E1 -26313.978,E2 -26313.978} C_VEL
LIN {X 0,Y 134.222,Z 453.356,A -85,B 0,C 180,E1 -26318.927,E2 -26318.927} C_VEL
LIN {X 0,Y 142.359,Z 454.741,A -85,B 0,C 180,E1 -26322.515,E2 -26322.515} C_VEL
LIN {X 0,Y 142.226,Z 454.933,A -85,B 0,C 180,E1 -26323.456,E2 -26323.456} C_VEL
LIN {X 0,Y 134.002,Z 455.047,A -85,B 0,C 180,E1 -26327.014,E2 -26327.014} C_VEL
LIN {X 0,Y 125.534,Z 454.467,A -85,B 0,C 180,E1 -26331.987,E2 -26331.987} C_VEL
LIN {X 0,Y 118.471,Z 453.045,A -85,B 0,C 180,E1 -26337.73,E2 -26337.73} C_VEL
LIN {X 0,Y 112.533,Z 450.672,A -85,B 0,C 180,E1 -26345.067,E2 -26345.067} C_VEL
LIN {X 0,Y 108.68,Z 455.052,A -85,B 0,C 180,E1 -26351.135,E2 -26351.135} C_VEL
LIN {X 0,Y 107.257,Z 456.959,A -85,B 0,C 180,E1 -26354.805,E2 -26354.805} C_VEL
LIN {X 0,Y 106.286,Z 458.403,A -85,B 0,C 180,E1 -26358.558,E2 -26358.558} C_VEL
LIN {X 0,Y 105.574,Z 460.069,A -85,B 0,C 180,E1 -26366.183,E2 -26366.183} C_VEL
LIN {X 0,Y 105.747,Z 460.303,A -85,B 0,C 180,E1 -26370,E2 -26370} C_VEL
LIN {X 0,Y 105.501,Z 460.049,A -85,B 0,C 180,E1 -26373.82,E2 -26373.82} C_VEL
LIN {X 0,Y 105.525,Z 459.395,A -85,B 0,C 180,E1 -26377.655,E2 -26377.655} C_VEL
LIN {X 0,Y 105.915,Z 458.347,A -85,B 0,C 180,E1 -26381.482,E2 -26381.482} C_VEL
LIN {X 0,Y 106.749,Z 456.875,A -85,B 0,C 180,E1 -26385.269,E2 -26385.269} C_VEL
LIN {X 0,Y 108.782,Z 453.842,A -85,B 0,C 180,E1 -26390.814,E2 -26390.814} C_VEL
LIN {X 0,Y 112.066,Z 449.769,A -85,B 0,C 180,E1 -26396.04,E2 -26396.04} C_VEL
LIN {X 0,Y 117.189,Z 443.522,A -85,B 0,C 180,E1 -26401.652,E2 -26401.652} C_VEL
LIN {X 0,Y 118.518,Z 442.267,A -85,B 0,C 180,E1 -26402.759,E2 -26402.759} C_VEL
LIN {X 0,Y 124.904,Z 443.058,A -85,B 0,C 180,E1 -26408.239,E2 -26408.239} C_VEL
LIN {X 0,Y 133.247,Z 443.163,A -85,B 0,C 180,E1 -26413.289,E2 -26413.289} C_VEL
LIN {X 0,Y 142.836,Z 442.52,A -85,B 0,C 180,E1 -26417.566,E2 -26417.566} C_VEL
LIN {X 0,Y 143.935,Z 442.198,A -85,B 0,C 180,E1 -26418.633,E2 -26418.633} C_VEL
LIN {X 0,Y 136.439,Z 440.791,A -85,B 0,C 180,E1 -26421.821,E2 -26421.821} C_VEL
LIN {X 0,Y 127.672,Z 437.948,A -85,B 0,C 180,E1 -26426.601,E2 -26426.601} C_VEL
LIN {X 0,Y 120.346,Z 433.987,A -85,B 0,C 180,E1 -26432.148,E2 -26432.148} C_VEL
LIN {X 0,Y 114.542,Z 428.811,A -85,B 0,C 180,E1 -26438.399,E2 -26438.399} C_VEL
LIN {X 0,Y 112.948,Z 426.798,A -85,B 0,C 180,E1 -26440.633,E2 -26440.633} C_VEL
LIN {X 0,Y 110.763,Z 424.232,A -85,B 0,C 180,E1 -26443.093,E2 -26443.093} C_VEL
LIN {X 0,Y 106.025,Z 419.304,A -85,B 0,C 180,E1 -26446.887,E2 -26446.887} C_VEL
LIN {X 0,Y 101.854,Z 413.792,A -85,B 0,C 180,E1 -26450.867,E2 -26450.867} C_VEL
LIN {X 0,Y 100.667,Z 410.36,A -85,B 0,C 180,E1 -26453.541,E2 -26453.541} C_VEL
LIN {X 0,Y 100.226,Z 403.083,A -85,B 0,C 180,E1 -26459.247,E2 -26459.247} C_VEL
LIN {X 0,Y 100.049,Z 403.233,A -85,B 0,C 180,E1 -26460,E2 -26460} C_VEL
LIN {X 0,Y 100.803,Z 402.132,A -85,B 0,C 180,E1 -26463.998,E2 -26463.998} C_VEL
LIN {X 0,Y 101.829,Z 400.885,A -85,B 0,C 180,E1 -26465.943,E2 -26465.943} C_VEL
LIN {X 0,Y 103.229,Z 399.259,A -85,B 0,C 180,E1 -26467.826,E2 -26467.826} C_VEL
LIN {X 0,Y 106.291,Z 397.008,A -85,B 0,C 180,E1 -26473.381,E2 -26473.381} C_VEL
LIN {X 0,Y 109.302,Z 394.179,A -85,B 0,C 180,E1 -26476.151,E2 -26476.151} C_VEL
LIN {X 0,Y 112.993,Z 391.818,A -85,B 0,C 180,E1 -26480.005,E2 -26480.005} C_VEL
LIN {X 0,Y 116.018,Z 389.45,A -85,B 0,C 180,E1 -26482.248,E2 -26482.248} C_VEL
LIN {X 0,Y 119.787,Z 385.902,A -85,B 0,C 180,E1 -26484.249,E2 -26484.249} C_VEL
LIN {X 0,Y 123.832,Z 383.333,A -85,B 0,C 180,E1 -26487.003,E2 -26487.003} C_VEL
LIN {X 0,Y 126.321,Z 381.23,A -85,B 0,C 180,E1 -26488.224,E2 -26488.224} C_VEL
LIN {X 0,Y 128.368,Z 380.243,A -85,B 0,C 180,E1 -26489.521,E2 -26489.521} C_VEL
LIN {X 0,Y 130.149,Z 386.305,A -85,B 0,C 180,E1 -26493.721,E2 -26493.721} C_VEL
LIN {X 0,Y 131.512,Z 393.271,A -85,B 0,C 180,E1 -26497.918,E2 -26497.918} C_VEL
LIN {X 0,Y 131.702,Z 396.832,A -85,B 0,C 180,E1 -26499.819,E2 -26499.819} C_VEL
LIN {X 0,Y 130.586,Z 404.612,A -85,B 0,C 180,E1 -26503.401,E2 -26503.401} C_VEL
LIN {X 0,Y 130.146,Z 406.613,A -85,B 0,C 180,E1 -26504.315,E2 -26504.315} C_VEL
LIN {X 0,Y 125.081,Z 415.518,A -85,B 0,C 180,E1 -26507.604,E2 -26507.604} C_VEL
LIN {X 0,Y 119.07,Z 424.215,A -85,B 0,C 180,E1 -26511.702,E2 -26511.702} C_VEL
LIN {X 0,Y 113.844,Z 431.161,A -85,B 0,C 180,E1 -26516.248,E2 -26516.248} C_VEL
LIN {X 0,Y 109.185,Z 436.681,A -85,B 0,C 180,E1 -26521.134,E2 -26521.134} C_VEL
LIN {X 0,Y 105.358,Z 441.002,A -85,B 0,C 180,E1 -26526.407,E2 -26526.407} C_VEL
LIN {X 0,Y 103.306,Z 443.271,A -85,B 0,C 180,E1 -26530.114,E2 -26530.114} C_VEL
LIN {X 0,Y 101.677,Z 445.115,A -85,B 0,C 180,E1 -26533.949,E2 -26533.949} C_VEL
LIN {X 0,Y 99.813,Z 447.183,A -85,B 0,C 180,E1 -26540.324,E2 -26540.324} C_VEL
LIN {X 0,Y 98.945,Z 448.104,A -85,B 0,C 180,E1 -26545.927,E2 -26545.927} C_VEL
LIN {X 0,Y 98.783,Z 448.329,A -85,B 0,C 180,E1 -26550,E2 -26550} C_VEL
LIN {X 0,Y 98.94,Z 448.13,A -85,B 0,C 180,E1 -26554.073,E2 -26554.073} C_VEL
LIN {X 0,Y 99.627,Z 447.37,A -85,B 0,C 180,E1 -26559.029,E2 -26559.029} C_VEL
LIN {X 0,Y 101.608,Z 445.214,A -85,B 0,C 180,E1 -26566.062,E2 -26566.062} C_VEL
LIN {X 0,Y 104.227,Z 442.345,A -85,B 0,C 180,E1 -26571.769,E2 -26571.769} C_VEL
LIN {X 0,Y 107.767,Z 438.435,A -85,B 0,C 180,E1 -26577.162,E2 -26577.162} C_VEL
LIN {X 0,Y 112.126,Z 433.359,A -85,B 0,C 180,E1 -26582.193,E2 -26582.193} C_VEL
LIN {X 0,Y 117.154,Z 426.955,A -85,B 0,C 180,E1 -26586.863,E2 -26586.863} C_VEL
LIN {X 0,Y 122.967,Z 418.973,A -85,B 0,C 180,E1 -26591.092,E2 -26591.092} C_VEL
LIN {X 0,Y 128.102,Z 410.634,A -85,B 0,C 180,E1 -26594.503,E2 -26594.503} C_VEL
LIN {X 0,Y 130.078,Z 407.05,A -85,B 0,C 180,E1 -26595.716,E2 -26595.716} C_VEL
LIN {X 0,Y 130.973,Z 403.053,A -85,B 0,C 180,E1 -26597.546,E2 -26597.546} C_VEL
LIN {X 0,Y 131.858,Z 396.098,A -85,B 0,C 180,E1 -26600.733,E2 -26600.733} C_VEL
LIN {X 0,Y 131.277,Z 391.362,A -85,B 0,C 180,E1 -26603.421,E2 -26603.421} C_VEL
LIN {X 0,Y 129.943,Z 385.229,A -85,B 0,C 180,E1 -26607.258,E2 -26607.258} C_VEL
LIN {X 0,Y 125.688,Z 386.825,A -85,B 0,C 180,E1 -26609.785,E2 -26609.785} C_VEL
LIN {X 0,Y 121.2,Z 389.403,A -85,B 0,C 180,E1 -26612.361,E2 -26612.361} C_VEL
LIN {X 0,Y 116.086,Z 393.418,A -85,B 0,C 180,E1 -26614.926,E2 -26614.926} C_VEL
LIN {X 0,Y 112.533,Z 395.102,A -85,B 0,C 180,E1 -26617.993,E2 -26617.993} C_VEL
LIN {X 0,Y 108.077,Z 398.635,A -85,B 0,C 180,E1 -26621.026,E2 -26621.026} C_VEL
LIN {X 0,Y 103.949,Z 401.048,A -85,B 0,C 180,E1 -26626.165,E2 -26626.165} C_VEL
LIN {X 0,Y 102.08,Z 402.68,A -85,B 0,C 180,E1 -26628.08,E2 -26628.08} C_VEL
LIN {X 0,Y 100.463,Z 403.608,A -85,B 0,C 180,E1 -26631.957,E2 -26631.957} C_VEL
LIN {X 0,Y 100.617,Z 403.288,A -85,B 0,C 180,E1 -26632.6,E2 -26632.6} C_VEL
LIN {X 0,Y 100.278,Z 412.477,A -85,B 0,C 180,E1 -26637.992,E2 -26637.992} C_VEL
LIN {X 0,Y 100.411,Z 419.72,A -85,B 0,C 180,E1 -26643.009,E2 -26643.009} C_VEL
LIN {X 0,Y 101.116,Z 427.028,A -85,B 0,C 180,E1 -26648.997,E2 -26648.997} C_VEL
LIN {X 0,Y 102.814,Z 434.067,A -85,B 0,C 180,E1 -26655.868,E2 -26655.868} C_VEL
LIN {X 0,Y 106.749,Z 440.665,A -85,B 0,C 180,E1 -26663.267,E2 -26663.267} C_VEL
LIN {X 0,Y 112.509,Z 445.956,A -85,B 0,C 180,E1 -26669.982,E2 -26669.982} C_VEL
LIN {X 0,Y 119.958,Z 450.092,A -85,B 0,C 180,E1 -26675.865,E2 -26675.865} C_VEL
LIN {X 0,Y 128.782,Z 453.114,A -85,B 0,C 180,E1 -26680.91,E2 -26680.91} C_VEL
LIN {X 0,Y 132.228,Z 453.939,A -85,B 0,C 180,E1 -26682.479,E2 -26682.479} C_VEL
LIN {X 0,Y 131.069,Z 454.09,A -85,B 0,C 180,E1 -26683.915,E2 -26683.915} C_VEL
LIN {X 0,Y 120.128,Z 453.033,A -85,B 0,C 180,E1 -26689.943,E2 -26689.943} C_VEL
LIN {X 0,Y 112.704,Z 451.281,A -85,B 0,C 180,E1 -26695.859,E2 -26695.859} C_VEL
LIN {X 0,Y 107.39,Z 449.035,A -85,B 0,C 180,E1 -26702.074,E2 -26702.074} C_VEL
LIN {X 0,Y 102.974,Z 453.553,A -85,B 0,C 180,E1 -26707.952,E2 -26707.952} C_VEL
LIN {X 0,Y 100.41,Z 456.544,A -85,B 0,C 180,E1 -26713.741,E2 -26713.741} C_VEL
LIN {X 0,Y 99.32,Z 457.987,A -85,B 0,C 180,E1 -26717.744,E2 -26717.744} C_VEL
LIN {X 0,Y 98.493,Z 459.653,A -85,B 0,C 180,E1 -26725.908,E2 -26725.908} C_VEL
LIN {X 0,Y 98.647,Z 459.888,A -85,B 0,C 180,E1 -26730,E2 -26730} C_VEL
LIN {X 0,Y 98.401,Z 459.633,A -85,B 0,C 180,E1 -26734.096,E2 -26734.096} C_VEL
LIN {X 0,Y 98.483,Z 458.979,A -85,B 0,C 180,E1 -26738.206,E2 -26738.206} C_VEL
LIN {X 0,Y 98.939,Z 457.929,A -85,B 0,C 180,E1 -26742.304,E2 -26742.304} C_VEL
LIN {X 0,Y 99.862,Z 456.456,A -85,B 0,C 180,E1 -26746.35,E2 -26746.35} C_VEL
LIN {X 0,Y 102.166,Z 453.426,A -85,B 0,C 180,E1 -26752.231,E2 -26752.231} C_VEL
LIN {X 0,Y 105.733,Z 449.354,A -85,B 0,C 180,E1 -26757.729,E2 -26757.729} C_VEL
LIN {X 0,Y 110.337,Z 444.113,A -85,B 0,C 180,E1 -26762.78,E2 -26762.78} C_VEL
LIN {X 0,Y 113.627,Z 440.526,A -85,B 0,C 180,E1 -26765.441,E2 -26765.441} C_VEL
LIN {X 0,Y 123.721,Z 441.736,A -85,B 0,C 180,E1 -26772.974,E2 -26772.974} C_VEL
LIN {X 0,Y 133.085,Z 441.825,A -85,B 0,C 180,E1 -26777.674,E2 -26777.674} C_VEL
LIN {X 0,Y 133.718,Z 441.576,A -85,B 0,C 180,E1 -26778.677,E2 -26778.677} C_VEL
LIN {X 0,Y 126.189,Z 439.357,A -85,B 0,C 180,E1 -26782.22,E2 -26782.22} C_VEL
LIN {X 0,Y 117.832,Z 435.555,A -85,B 0,C 180,E1 -26787.534,E2 -26787.534} C_VEL
LIN {X 0,Y 110.883,Z 430.614,A -85,B 0,C 180,E1 -26793.662,E2 -26793.662} C_VEL
LIN {X 0,Y 105.629,Z 424.381,A -85,B 0,C 180,E1 -26800.569,E2 -26800.569} C_VEL
LIN {X 0,Y 102.082,Z 416.677,A -85,B 0,C 180,E1 -26808.081,E2 -26808.081} C_VEL
LIN {X 0,Y 100.667,Z 410.36,A -85,B 0,C 180,E1 -26813.541,E2 -26813.541} C_VEL
LIN {X 0,Y 100.067,Z 407.756,A -85,B 0,C 180,E1 -26816.495,E2 -26816.495} C_VEL
LIN {X 0,Y 99.374,Z 406.294,A -85,B 0,C 180,E1 -26819.743,E2 -26819.743} C_VEL
LIN {X 0,Y 99.018,Z 405.089,A -85,B 0,C 180,E1 -26826.634,E2 -26826.634} C_VEL
LIN {X 0,Y 100.437,Z 404.091,A -85,B 0,C 180,E1 -26831.132,E2 -26831.132} C_VEL
LIN {X 0,Y 103.648,Z 401.994,A -85,B 0,C 180,E1 -26835.738,E2 -26835.738} C_VEL
LIN {X 0,Y 107.568,Z 398.92,A -85,B 0,C 180,E1 -26839.067,E2 -26839.067} C_VEL
LIN {X 0,Y 111.058,Z 396.966,A -85,B 0,C 180,E1 -26842.315,E2 -26842.315} C_VEL
LIN {X 0,Y 113.175,Z 395.592,A -85,B 0,C 180,E1 -26843.806,E2 -26843.806} C_VEL
LIN {X 0,Y 118.382,Z 391.294,A -85,B 0,C 180,E1 -26846.438,E2 -26846.438} C_VEL
LIN {X 0,Y 122.807,Z 388.698,A -85,B 0,C 180,E1 -26849.107,E2 -26849.107} C_VEL
LIN {X 0,Y 124.813,Z 387.968,A -85,B 0,C 180,E1 -26850.45,E2 -26850.45} C_VEL
LIN {X 0,Y 125.927,Z 394.018,A -85,B 0,C 180,E1 -26854.639,E2 -26854.639} C_VEL
LIN {X 0,Y 126.384,Z 398.878,A -85,B 0,C 180,E1 -26857.712,E2 -26857.712} C_VEL
LIN {X 0,Y 125.387,Z 405.059,A -85,B 0,C 180,E1 -26860.827,E2 -26860.827} C_VEL
LIN {X 0,Y 124.938,Z 407.054,A -85,B 0,C 180,E1 -26861.812,E2 -26861.812} C_VEL
LIN {X 0,Y 124.17,Z 408.93,A -85,B 0,C 180,E1 -26862.625,E2 -26862.625} C_VEL
LIN {X 0,Y 118.867,Z 417.524,A -85,B 0,C 180,E1 -26865.995,E2 -26865.995} C_VEL
LIN {X 0,Y 113.605,Z 424.627,A -85,B 0,C 180,E1 -26869.491,E2 -26869.491} C_VEL
LIN {X 0,Y 108.003,Z 431.577,A -85,B 0,C 180,E1 -26874.151,E2 -26874.151} C_VEL
LIN {X 0,Y 103.045,Z 437.095,A -85,B 0,C 180,E1 -26879.235,E2 -26879.235} C_VEL
LIN {X 0,Y 98.909,Z 441.417,A -85,B 0,C 180,E1 -26884.765,E2 -26884.765} C_VEL
LIN {X 0,Y 96.669,Z 443.686,A -85,B 0,C 180,E1 -26888.684,E2 -26888.684} C_VEL
LIN {X 0,Y 94.875,Z 445.531,A -85,B 0,C 180,E1 -26892.764,E2 -26892.764} C_VEL
LIN {X 0,Y 92.693,Z 447.738,A -85,B 0,C 180,E1 -26900.289,E2 -26900.289} C_VEL
LIN {X 0,Y 91.877,Z 448.519,A -85,B 0,C 180,E1 -26905.613,E2 -26905.613} C_VEL
LIN {X 0,Y 91.695,Z 448.744,A -85,B 0,C 180,E1 -26910,E2 -26910} C_VEL
LIN {X 0,Y 91.891,Z 448.544,A -85,B 0,C 180,E1 -26914.386,E2 -26914.386} C_VEL
LIN {X 0,Y 92.55,Z 447.879,A -85,B 0,C 180,E1 -26919.181,E2 -26919.181} C_VEL
LIN {X 0,Y 94.824,Z 445.628,A -85,B 0,C 180,E1 -26927.245,E2 -26927.245} C_VEL
LIN {X 0,Y 97.683,Z 442.758,A -85,B 0,C 180,E1 -26933.31,E2 -26933.31} C_VEL
LIN {X 0,Y 101.518,Z 438.847,A -85,B 0,C 180,E1 -26938.987,E2 -26938.987} C_VEL
LIN {X 0,Y 106.203,Z 433.769,A -85,B 0,C 180,E1 -26944.228,E2 -26944.228} C_VEL
LIN {X 0,Y 111.571,Z 427.364,A -85,B 0,C 180,E1 -26949.044,E2 -26949.044} C_VEL
LIN {X 0,Y 117.724,Z 419.38,A -85,B 0,C 180,E1 -26953.357,E2 -26953.357} C_VEL
LIN {X 0,Y 123.468,Z 410.494,A -85,B 0,C 180,E1 -26957.013,E2 -26957.013} C_VEL
LIN {X 0,Y 124.976,Z 407.475,A -85,B 0,C 180,E1 -26958.169,E2 -26958.169} C_VEL
LIN {X 0,Y 126.446,Z 399.886,A -85,B 0,C 180,E1 -26961.945,E2 -26961.945} C_VEL
LIN {X 0,Y 126.278,Z 396.081,A -85,B 0,C 180,E1 -26964.241,E2 -26964.241} C_VEL
LIN {X 0,Y 125.901,Z 393.334,A -85,B 0,C 180,E1 -26966.067,E2 -26966.067} C_VEL
LIN {X 0,Y 124.629,Z 392.295,A -85,B 0,C 180,E1 -26967.607,E2 -26967.607} C_VEL
LIN {X 0,Y 119.92,Z 394.674,A -85,B 0,C 180,E1 -26970.122,E2 -26970.122} C_VEL
LIN {X 0,Y 114.096,Z 398.73,A -85,B 0,C 180,E1 -26972.8,E2 -26972.8} C_VEL
LIN {X 0,Y 110.507,Z 400.31,A -85,B 0,C 180,E1 -26975.582,E2 -26975.582} C_VEL
LIN {X 0,Y 105.621,Z 403.657,A -85,B 0,C 180,E1 -26978.68,E2 -26978.68} C_VEL
LIN {X 0,Y 100.861,Z 406.194,A -85,B 0,C 180,E1 -26983.816,E2 -26983.816} C_VEL
LIN {X 0,Y 99.075,Z 407.464,A -85,B 0,C 180,E1 -26985.624,E2 -26985.624} C_VEL
LIN {X 0,Y 97.745,Z 408.297,A -85,B 0,C 180,E1 -26987.543,E2 -26987.543} C_VEL
LIN {X 0,Y 95.924,Z 409.362,A -85,B 0,C 180,E1 -26991.574,E2 -26991.574} C_VEL
LIN {X 0,Y 94.489,Z 410.746,A -85,B 0,C 180,E1 -26993.594,E2 -26993.594} C_VEL
LIN {X 0,Y 93.546,Z 411.642,A -85,B 0,C 180,E1 -26995.691,E2 -26995.691} C_VEL
LIN {X 0,Y 93.183,Z 412.023,A -85,B 0,C 180,E1 -26997.839,E2 -26997.839} C_VEL
LIN {X 0,Y 93.561,Z 411.885,A -85,B 0,C 180,E1 -26999.596,E2 -26999.596} C_VEL
LIN {X 0,Y 93.774,Z 418.312,A -85,B 0,C 180,E1 -27004.298,E2 -27004.298} C_VEL
LIN {X 0,Y 94.901,Z 426.864,A -85,B 0,C 180,E1 -27011.751,E2 -27011.751} C_VEL
LIN {X 0,Y 96.893,Z 433.371,A -85,B 0,C 180,E1 -27018.472,E2 -27018.472} C_VEL
LIN {X 0,Y 101.813,Z 440.582,A -85,B 0,C 180,E1 -27026.659,E2 -27026.659} C_VEL
LIN {X 0,Y 108.301,Z 445.938,A -85,B 0,C 180,E1 -27033.476,E2 -27033.476} C_VEL
LIN {X 0,Y 114.322,Z 449.195,A -85,B 0,C 180,E1 -27037.934,E2 -27037.934} C_VEL
LIN {X 0,Y 122.314,Z 452.276,A -85,B 0,C 180,E1 -27042.465,E2 -27042.465} C_VEL
LIN {X 0,Y 121.124,Z 452.344,A -85,B 0,C 180,E1 -27044.129,E2 -27044.129} C_VEL
LIN {X 0,Y 110.847,Z 450.43,A -85,B 0,C 180,E1 -27050.652,E2 -27050.652} C_VEL
LIN {X 0,Y 102.613,Z 447.319,A -85,B 0,C 180,E1 -27058.805,E2 -27058.805} C_VEL
LIN {X 0,Y 97.668,Z 451.897,A -85,B 0,C 180,E1 -27064.421,E2 -27064.421} C_VEL
LIN {X 0,Y 95.332,Z 454.222,A -85,B 0,C 180,E1 -27068.37,E2 -27068.37} C_VEL
LIN {X 0,Y 93.611,Z 456.129,A -85,B 0,C 180,E1 -27072.524,E2 -27072.524} C_VEL
LIN {X 0,Y 92.392,Z 457.571,A -85,B 0,C 180,E1 -27076.809,E2 -27076.809} C_VEL
LIN {X 0,Y 91.399,Z 459.237,A -85,B 0,C 180,E1 -27085.59,E2 -27085.59} C_VEL
LIN {X 0,Y 91.545,Z 459.472,A -85,B 0,C 180,E1 -27090,E2 -27090} C_VEL
LIN {X 0,Y 91.309,Z 459.216,A -85,B 0,C 180,E1 -27094.414,E2 -27094.414} C_VEL
LIN {X 0,Y 91.996,Z 457.512,A -85,B 0,C 180,E1 -27103.249,E2 -27103.249} C_VEL
LIN {X 0,Y 93.026,Z 456.037,A -85,B 0,C 180,E1 -27107.59,E2 -27107.59} C_VEL
LIN {X 0,Y 95.6,Z 453.008,A -85,B 0,C 180,E1 -27113.849,E2 -27113.849} C_VEL
LIN {X 0,Y 99.505,Z 448.938,A -85,B 0,C 180,E1 -27119.631,E2 -27119.631} C_VEL
LIN {X 0,Y 104.442,Z 443.698,A -85,B 0,C 180,E1 -27124.888,E2 -27124.888} C_VEL
LIN {X 0,Y 109.263,Z 438.676,A -85,B 0,C 180,E1 -27128.544,E2 -27128.544} C_VEL
LIN {X 0,Y 118.758,Z 440.046,A -85,B 0,C 180,E1 -27135.247,E2 -27135.247} C_VEL
LIN {X 0,Y 123.494,Z 440.37,A -85,B 0,C 180,E1 -27137.717,E2 -27137.717} C_VEL
LIN {X 0,Y 120.667,Z 438.987,A -85,B 0,C 180,E1 -27140.158,E2 -27140.158} C_VEL
LIN {X 0,Y 111.936,Z 434.789,A -85,B 0,C 180,E1 -27145.593,E2 -27145.593} C_VEL
LIN {X 0,Y 104.664,Z 429.435,A -85,B 0,C 180,E1 -27151.963,E2 -27151.963} C_VEL
LIN {X 0,Y 99.107,Z 422.801,A -85,B 0,C 180,E1 -27159.233,E2 -27159.233} C_VEL
LIN {X 0,Y 95.369,Z 414.695,A -85,B 0,C 180,E1 -27167.228,E2 -27167.228} C_VEL
LIN {X 0,Y 94.882,Z 412.996,A -85,B 0,C 180,E1 -27168.788,E2 -27168.788} C_VEL
LIN {X 0,Y 93.942,Z 412.941,A -85,B 0,C 180,E1 -27171.395,E2 -27171.395} C_VEL
LIN {X 0,Y 94.109,Z 411.435,A -85,B 0,C 180,E1 -27175.717,E2 -27175.717} C_VEL
LIN {X 0,Y 95.684,Z 408.823,A -85,B 0,C 180,E1 -27180,E2 -27180} C_VEL
LIN {X 0,Y 96.432,Z 407.83,A -85,B 0,C 180,E1 -27184.18,E2 -27184.18} C_VEL
LIN {X 0,Y 97.275,Z 406.995,A -85,B 0,C 180,E1 -27186.222,E2 -27186.222} C_VEL
LIN {X 0,Y 100.011,Z 404.379,A -85,B 0,C 180,E1 -27190.323,E2 -27190.323} C_VEL
LIN {X 0,Y 100.437,Z 404.091,A -85,B 0,C 180,E1 -27191.132,E2 -27191.132} C_VEL
LIN {X 0,Y 101.686,Z 403.668,A -85,B 0,C 180,E1 -27194.069,E2 -27194.069} C_VEL
LIN {X 0,Y 104.52,Z 404.019,A -85,B 0,C 180,E1 -27200.592,E2 -27200.592} C_VEL
LIN {X 0,Y 106.241,Z 403.392,A -85,B 0,C 180,E1 -27202.508,E2 -27202.508} C_VEL
LIN {X 0,Y 109.063,Z 401.94,A -85,B 0,C 180,E1 -27204.763,E2 -27204.763} C_VEL
LIN {X 0,Y 111.371,Z 400.58,A -85,B 0,C 180,E1 -27206.215,E2 -27206.215} C_VEL
LIN {X 0,Y 116.924,Z 396.48,A -85,B 0,C 180,E1 -27208.742,E2 -27208.742} C_VEL
LIN {X 0,Y 119.291,Z 395.217,A -85,B 0,C 180,E1 -27210.052,E2 -27210.052} C_VEL
LIN {X 0,Y 120.636,Z 395.782,A -85,B 0,C 180,E1 -27211.623,E2 -27211.623} C_VEL
LIN {X 0,Y 121.015,Z 401.905,A -85,B 0,C 180,E1 -27215.964,E2 -27215.964} C_VEL
LIN {X 0,Y 120.235,Z 406.146,A -85,B 0,C 180,E1 -27218.322,E2 -27218.322} C_VEL
LIN {X 0,Y 119.338,Z 409.353,A -85,B 0,C 180,E1 -27220.04,E2 -27220.04} C_VEL
LIN {X 0,Y 115.017,Z 416.341,A -85,B 0,C 180,E1 -27222.84,E2 -27222.84} C_VEL
LIN {X 0,Y 108.328,Z 425.039,A -85,B 0,C 180,E1 -27227.062,E2 -27227.062} C_VEL
LIN {X 0,Y 102.327,Z 431.992,A -85,B 0,C 180,E1 -27231.82,E2 -27231.82} C_VEL
LIN {X 0,Y 97.037,Z 437.509,A -85,B 0,C 180,E1 -27237.098,E2 -27237.098} C_VEL
LIN {X 0,Y 92.559,Z 441.831,A -85,B 0,C 180,E1 -27242.898,E2 -27242.898} C_VEL
LIN {X 0,Y 90.091,Z 444.102,A -85,B 0,C 180,E1 -27247.042,E2 -27247.042} C_VEL
LIN {X 0,Y 88.137,Z 445.946,A -85,B 0,C 180,E1 -27251.4,E2 -27251.4} C_VEL
LIN {X 0,Y 86.614,Z 447.345,A -85,B 0,C 180,E1 -27255.911,E2 -27255.911} C_VEL
LIN {X 0,Y 85.5,Z 448.328,A -85,B 0,C 180,E1 -27260.538,E2 -27260.538} C_VEL
LIN {X 0,Y 84.61,Z 449.159,A -85,B 0,C 180,E1 -27270,E2 -27270} C_VEL
LIN {X 0,Y 84.824,Z 448.959,A -85,B 0,C 180,E1 -27274.753,E2 -27274.753} C_VEL
LIN {X 0,Y 85.5,Z 448.37,A -85,B 0,C 180,E1 -27279.462,E2 -27279.462} C_VEL
LIN {X 0,Y 86.561,Z 447.407,A -85,B 0,C 180,E1 -27284.098,E2 -27284.098} C_VEL
LIN {X 0,Y 88.068,Z 446.042,A -85,B 0,C 180,E1 -27288.615,E2 -27288.615} C_VEL
LIN {X 0,Y 91.228,Z 443.171,A -85,B 0,C 180,E1 -27295.069,E2 -27295.069} C_VEL
LIN {X 0,Y 95.391,Z 439.259,A -85,B 0,C 180,E1 -27301.046,E2 -27301.046} C_VEL
LIN {X 0,Y 100.407,Z 434.181,A -85,B 0,C 180,E1 -27306.51,E2 -27306.51} C_VEL
LIN {X 0,Y 106.171,Z 427.773,A -85,B 0,C 180,E1 -27311.449,E2 -27311.449} C_VEL
LIN {X 0,Y 112.684,Z 419.787,A -85,B 0,C 180,E1 -27315.828,E2 -27315.828} C_VEL
LIN {X 0,Y 118.647,Z 411.045,A -85,B 0,C 180,E1 -27319.47,E2 -27319.47} C_VEL
LIN {X 0,Y 119.34,Z 409.772,A -85,B 0,C 180,E1 -27319.959,E2 -27319.959} C_VEL
LIN {X 0,Y 121.086,Z 403.145,A -85,B 0,C 180,E1 -27323.493,E2 -27323.493} C_VEL
LIN {X 0,Y 121.004,Z 398.717,A -85,B 0,C 180,E1 -27326.511,E2 -27326.511} C_VEL
LIN {X 0,Y 118.591,Z 399.73,A -85,B 0,C 180,E1 -27327.767,E2 -27327.767} C_VEL
LIN {X 0,Y 112.889,Z 403.31,A -85,B 0,C 180,E1 -27330.129,E2 -27330.129} C_VEL
LIN {X 0,Y 108.416,Z 405.303,A -85,B 0,C 180,E1 -27333.014,E2 -27333.014} C_VEL
LIN {X 0,Y 106.059,Z 406.576,A -85,B 0,C 180,E1 -27334.486,E2 -27334.486} C_VEL
LIN {X 0,Y 103.474,Z 408.244,A -85,B 0,C 180,E1 -27335.95,E2 -27335.95} C_VEL
LIN {X 0,Y 95.02,Z 412.658,A -85,B 0,C 180,E1 -27344.056,E2 -27344.056} C_VEL
LIN {X 0,Y 88.679,Z 416.845,A -85,B 0,C 180,E1 -27355.454,E2 -27355.454} C_VEL
LIN {X 0,Y 87.788,Z 417.86,A -85,B 0,C 180,E1 -27360,E2 -27360} C_VEL
LIN {X 0,Y 86.756,Z 419.58,A -85,B 0,C 180,E1 -27364.646,E2 -27364.646} C_VEL
LIN {X 0,Y 86.989,Z 419.904,A -85,B 0,C 180,E1 -27366.96,E2 -27366.96} C_VEL
LIN {X 0,Y 87.579,Z 419.869,A -85,B 0,C 180,E1 -27368.508,E2 -27368.508} C_VEL
LIN {X 0,Y 88.927,Z 426.586,A -85,B 0,C 180,E1 -27374.883,E2 -27374.883} C_VEL
LIN {X 0,Y 92.806,Z 435.239,A -85,B 0,C 180,E1 -27384.376,E2 -27384.376} C_VEL
LIN {X 0,Y 98.935,Z 441.803,A -85,B 0,C 180,E1 -27392.193,E2 -27392.193} C_VEL
LIN {X 0,Y 106.662,Z 446.962,A -85,B 0,C 180,E1 -27398.753,E2 -27398.753} C_VEL
LIN {X 0,Y 113.502,Z 450.158,A -85,B 0,C 180,E1 -27402.931,E2 -27402.931} C_VEL
LIN {X 0,Y 105.689,Z 448.394,A -85,B 0,C 180,E1 -27408.32,E2 -27408.32} C_VEL
LIN {X 0,Y 98.088,Z 445.607,A -85,B 0,C 180,E1 -27415.339,E2 -27415.339} C_VEL
LIN {X 0,Y 92.863,Z 450.144,A -85,B 0,C 180,E1 -27420.533,E2 -27420.533} C_VEL
LIN {X 0,Y 88.773,Z 453.808,A -85,B 0,C 180,E1 -27426.681,E2 -27426.681} C_VEL
LIN {X 0,Y 86.84,Z 455.713,A -85,B 0,C 180,E1 -27431.112,E2 -27431.112} C_VEL
LIN {X 0,Y 85.476,Z 457.155,A -85,B 0,C 180,E1 -27435.72,E2 -27435.72} C_VEL
LIN {X 0,Y 84.314,Z 458.821,A -85,B 0,C 180,E1 -27445.219,E2 -27445.219} C_VEL
LIN {X 0,Y 84.465,Z 459.057,A -85,B 0,C 180,E1 -27450,E2 -27450} C_VEL
LIN {X 0,Y 84.217,Z 458.799,A -85,B 0,C 180,E1 -27454.787,E2 -27454.787} C_VEL
LIN {X 0,Y 84.391,Z 458.143,A -85,B 0,C 180,E1 -27459.588,E2 -27459.588} C_VEL
LIN {X 0,Y 85.058,Z 457.094,A -85,B 0,C 180,E1 -27464.352,E2 -27464.352} C_VEL
LIN {X 0,Y 86.251,Z 455.619,A -85,B 0,C 180,E1 -27469.022,E2 -27469.022} C_VEL
LIN {X 0,Y 89.13,Z 452.59,A -85,B 0,C 180,E1 -27475.701,E2 -27475.701} C_VEL
LIN {X 0,Y 93.384,Z 448.521,A -85,B 0,C 180,E1 -27481.791,E2 -27481.791} C_VEL
LIN {X 0,Y 98.709,Z 443.284,A -85,B 0,C 180,E1 -27487.243,E2 -27487.243} C_VEL
LIN {X 0,Y 105.442,Z 436.732,A -85,B 0,C 180,E1 -27491.979,E2 -27491.979} C_VEL
LIN {X 0,Y 114.056,Z 438.146,A -85,B 0,C 180,E1 -27497.683,E2 -27497.683} C_VEL
LIN {X 0,Y 110.583,Z 436.217,A -85,B 0,C 180,E1 -27500.54,E2 -27500.54} C_VEL
LIN {X 0,Y 102.166,Z 431.059,A -85,B 0,C 180,E1 -27506.611,E2 -27506.611} C_VEL
LIN {X 0,Y 94.013,Z 422.919,A -85,B 0,C 180,E1 -27515.723,E2 -27515.723} C_VEL
LIN {X 0,Y 92.964,Z 421.714,A -85,B 0,C 180,E1 -27517.205,E2 -27517.205} C_VEL
LIN {X 0,Y 90.446,Z 420.998,A -85,B 0,C 180,E1 -27521.892,E2 -27521.892} C_VEL
LIN {X 0,Y 89.156,Z 418.103,A -85,B 0,C 180,E1 -27530.929,E2 -27530.929} C_VEL
LIN {X 0,Y 89.184,Z 416.828,A -85,B 0,C 180,E1 -27535.48,E2 -27535.48} C_VEL
LIN {X 0,Y 90.466,Z 414.78,A -85,B 0,C 180,E1 -27540,E2 -27540} C_VEL
LIN {X 0,Y 93.634,Z 411.658,A -85,B 0,C 180,E1 -27548.634,E2 -27548.634} C_VEL
LIN {X 0,Y 96.566,Z 409.381,A -85,B 0,C 180,E1 -27552.719,E2 -27552.719} C_VEL
LIN {X 0,Y 100.954,Z 406.774,A -85,B 0,C 180,E1 -27558.257,E2 -27558.257} C_VEL
LIN {X 0,Y 105.18,Z 403.939,A -85,B 0,C 180,E1 -27561.562,E2 -27561.562} C_VEL
LIN {X 0,Y 106.241,Z 403.392,A -85,B 0,C 180,E1 -27562.508,E2 -27562.508} C_VEL
LIN {X 0,Y 110.808,Z 401.331,A -85,B 0,C 180,E1 -27566.282,E2 -27566.282} C_VEL
LIN {X 0,Y 113.554,Z 400.745,A -85,B 0,C 180,E1 -27568.747,E2 -27568.747} C_VEL
LIN {X 0,Y 115.254,Z 401.336,A -85,B 0,C 180,E1 -27570.89,E2 -27570.89} C_VEL
LIN {X 0,Y 115.741,Z 402.642,A -85,B 0,C 180,E1 -27572.345,E2 -27572.345} C_VEL
LIN {X 0,Y 115.52,Z 406.385,A -85,B 0,C 180,E1 -27575.093,E2 -27575.093} C_VEL
LIN {X 0,Y 114.028,Z 411.239,A -85,B 0,C 180,E1 -27577.883,E2 -27577.883} C_VEL
LIN {X 0,Y 109.13,Z 418.347,A -85,B 0,C 180,E1 -27580.826,E2 -27580.826} C_VEL
LIN {X 0,Y 103.267,Z 425.451,A -85,B 0,C 180,E1 -27584.39,E2 -27584.39} C_VEL
LIN {X 0,Y 96.845,Z 432.407,A -85,B 0,C 180,E1 -27589.222,E2 -27589.222} C_VEL
LIN {X 0,Y 91.164,Z 437.924,A -85,B 0,C 180,E1 -27594.676,E2 -27594.676} C_VEL
LIN {X 0,Y 86.3,Z 442.247,A -85,B 0,C 180,E1 -27600.75,E2 -27600.75} C_VEL
LIN {X 0,Y 83.611,Z 444.517,A -85,B 0,C 180,E1 -27605.148,E2 -27605.148} C_VEL
LIN {X 0,Y 81.438,Z 446.362,A -85,B 0,C 180,E1 -27609.806,E2 -27609.806} C_VEL
LIN {X 0,Y 79.762,Z 447.76,A -85,B 0,C 180,E1 -27614.672,E2 -27614.672} C_VEL
LIN {X 0,Y 78.254,Z 448.958,A -85,B 0,C 180,E1 -27621.086,E2 -27621.086} C_VEL
LIN {X 0,Y 77.523,Z 449.574,A -85,B 0,C 180,E1 -27630,E2 -27630} C_VEL
LIN {X 0,Y 78.254,Z 449,A -85,B 0,C 180,E1 -27638.914,E2 -27638.914} C_VEL
LIN {X 0,Y 79.711,Z 447.82,A -85,B 0,C 180,E1 -27645.338,E2 -27645.338} C_VEL
LIN {X 0,Y 81.386,Z 446.456,A -85,B 0,C 180,E1 -27650.207,E2 -27650.207} C_VEL
LIN {X 0,Y 84.85,Z 443.585,A -85,B 0,C 180,E1 -27657.101,E2 -27657.101} C_VEL
LIN {X 0,Y 89.405,Z 439.67,A -85,B 0,C 180,E1 -27663.385,E2 -27663.385} C_VEL
LIN {X 0,Y 94.795,Z 434.593,A -85,B 0,C 180,E1 -27669.064,E2 -27669.064} C_VEL
LIN {X 0,Y 100.98,Z 428.181,A -85,B 0,C 180,E1 -27674.105,E2 -27674.105} C_VEL
LIN {X 0,Y 107.872,Z 420.194,A -85,B 0,C 180,E1 -27678.525,E2 -27678.525} C_VEL
LIN {X 0,Y 113.986,Z 411.689,A -85,B 0,C 180,E1 -27682.106,E2 -27682.106} C_VEL
LIN {X 0,Y 115.567,Z 406.917,A -85,B 0,C 180,E1 -27684.806,E2 -27684.806} C_VEL
LIN {X 0,Y 115.809,Z 405.627,A -85,B 0,C 180,E1 -27685.617,E2 -27685.617} C_VEL
LIN {X 0,Y 114.301,Z 406.194,A -85,B 0,C 180,E1 -27686.4,E2 -27686.4} C_VEL
LIN {X 0,Y 111.321,Z 407.956,A -85,B 0,C 180,E1 -27687.505,E2 -27687.505} C_VEL
LIN {X 0,Y 103.52,Z 411.373,A -85,B 0,C 180,E1 -27691.955,E2 -27691.955} C_VEL
LIN {X 0,Y 101.177,Z 412.734,A -85,B 0,C 180,E1 -27693.157,E2 -27693.157} C_VEL
LIN {X 0,Y 91.01,Z 417.482,A -85,B 0,C 180,E1 -27702.007,E2 -27702.007} C_VEL
LIN {X 0,Y 83.493,Z 421.811,A -85,B 0,C 180,E1 -27715.171,E2 -27715.171} C_VEL
LIN {X 0,Y 82.39,Z 422.951,A -85,B 0,C 180,E1 -27720,E2 -27720} C_VEL
LIN {X 0,Y 81.52,Z 424.374,A -85,B 0,C 180,E1 -27724.946,E2 -27724.946} C_VEL
LIN {X 0,Y 81.681,Z 425.409,A -85,B 0,C 180,E1 -27729.909,E2 -27729.909} C_VEL
LIN {X 0,Y 81.807,Z 426.998,A -85,B 0,C 180,E1 -27734.935,E2 -27734.935} C_VEL
LIN {X 0,Y 83.906,Z 427.997,A -85,B 0,C 180,E1 -27740.533,E2 -27740.533} C_VEL
LIN {X 0,Y 88.251,Z 434.971,A -85,B 0,C 180,E1 -27748.543,E2 -27748.543} C_VEL
LIN {X 0,Y 95.094,Z 441.458,A -85,B 0,C 180,E1 -27756.245,E2 -27756.245} C_VEL
LIN {X 0,Y 103.67,Z 446.782,A -85,B 0,C 180,E1 -27762.681,E2 -27762.681} C_VEL
LIN {X 0,Y 100.763,Z 446.107,A -85,B 0,C 180,E1 -27765.774,E2 -27765.774} C_VEL
LIN {X 0,Y 94.132,Z 443.737,A -85,B 0,C 180,E1 -27771.468,E2 -27771.468} C_VEL
LIN {X 0,Y 88.521,Z 448.294,A -85,B 0,C 180,E1 -27776.237,E2 -27776.237} C_VEL
LIN {X 0,Y 83.618,Z 452.311,A -85,B 0,C 180,E1 -27782.466,E2 -27782.466} C_VEL
LIN {X 0,Y 80.142,Z 455.298,A -85,B 0,C 180,E1 -27789.465,E2 -27789.465} C_VEL
LIN {X 0,Y 78.609,Z 456.74,A -85,B 0,C 180,E1 -27794.442,E2 -27794.442} C_VEL
LIN {X 0,Y 77.231,Z 458.405,A -85,B 0,C 180,E1 -27804.779,E2 -27804.779} C_VEL
LIN {X 0,Y 77.312,Z 458.624,A -85,B 0,C 180,E1 -27810.588,E2 -27810.588} C_VEL
LIN {X 0,Y 77.37,Z 457.725,A -85,B 0,C 180,E1 -27820.467,E2 -27820.467} C_VEL
LIN {X 0,Y 78.17,Z 456.676,A -85,B 0,C 180,E1 -27825.648,E2 -27825.648} C_VEL
LIN {X 0,Y 79.548,Z 455.201,A -85,B 0,C 180,E1 -27830.695,E2 -27830.695} C_VEL
LIN {X 0,Y 82.772,Z 452.173,A -85,B 0,C 180,E1 -27837.84,E2 -27837.84} C_VEL
LIN {X 0,Y 87.402,Z 448.104,A -85,B 0,C 180,E1 -27844.255,E2 -27844.255} C_VEL
LIN {X 0,Y 93.166,Z 442.869,A -85,B 0,C 180,E1 -27849.882,E2 -27849.882} C_VEL
LIN {X 0,Y 100.093,Z 436.322,A -85,B 0,C 180,E1 -27854.6,E2 -27854.6} C_VEL
LIN {X 0,Y 101.907,Z 434.641,A -85,B 0,C 180,E1 -27855.542,E2 -27855.542} C_VEL
LIN {X 0,Y 104.805,Z 435.211,A -85,B 0,C 180,E1 -27857.531,E2 -27857.531} C_VEL
LIN {X 0,Y 105.224,Z 435.206,A -85,B 0,C 180,E1 -27858.094,E2 -27858.094} C_VEL
LIN {X 0,Y 95.917,Z 429.343,A -85,B 0,C 180,E1 -27864.759,E2 -27864.759} C_VEL
LIN {X 0,Y 92.536,Z 428.954,A -85,B 0,C 180,E1 -27867.884,E2 -27867.884} C_VEL
LIN {X 0,Y 89.634,Z 427.942,A -85,B 0,C 180,E1 -27871.937,E2 -27871.937} C_VEL
LIN {X 0,Y 87.738,Z 426.446,A -85,B 0,C 180,E1 -27876.39,E2 -27876.39} C_VEL
LIN {X 0,Y 85.441,Z 425.793,A -85,B 0,C 180,E1 -27880.791,E2 -27880.791} C_VEL
LIN {X 0,Y 84.396,Z 421.068,A -85,B 0,C 180,E1 -27897.847,E2 -27897.847} C_VEL
LIN {X 0,Y 86.805,Z 418.406,A -85,B 0,C 180,E1 -27904.644,E2 -27904.644} C_VEL
LIN {X 0,Y 89.945,Z 416.098,A -85,B 0,C 180,E1 -27911.265,E2 -27911.265} C_VEL
LIN {X 0,Y 91.578,Z 414.987,A -85,B 0,C 180,E1 -27913.311,E2 -27913.311} C_VEL
LIN {X 0,Y 98.236,Z 411.356,A -85,B 0,C 180,E1 -27920.96,E2 -27920.96} C_VEL
LIN {X 0,Y 102.767,Z 408.748,A -85,B 0,C 180,E1 -27924.226,E2 -27924.226} C_VEL
LIN {X 0,Y 107.06,Z 406.701,A -85,B 0,C 180,E1 -27927.356,E2 -27927.356} C_VEL
LIN {X 0,Y 109.548,Z 405.365,A -85,B 0,C 180,E1 -27928.761,E2 -27928.761} C_VEL
LIN {X 0,Y 114.647,Z 402.024,A -85,B 0,C 180,E1 -27930.882,E2 -27930.882} C_VEL
LIN {X 0,Y 115.736,Z 401.904,A -85,B 0,C 180,E1 -27931.773,E2 -27931.773} C_VEL
LIN {X 0,Y 115.741,Z 402.642,A -85,B 0,C 180,E1 -27932.345,E2 -27932.345} C_VEL
LIN {X 0,Y 115.25,Z 404.712,A -85,B 0,C 180,E1 -27933.543,E2 -27933.543} C_VEL
LIN {X 0,Y 113.361,Z 408.14,A -85,B 0,C 180,E1 -27934.776,E2 -27934.776} C_VEL
LIN {X 0,Y 105.918,Z 417.165,A -85,B 0,C 180,E1 -27937.222,E2 -27937.222} C_VEL
LIN {X 0,Y 105.149,Z 418.102,A -85,B 0,C 180,E1 -27937.605,E2 -27937.605} C_VEL
LIN {X 0,Y 98.449,Z 425.864,A -85,B 0,C 180,E1 -27941.447,E2 -27941.447} C_VEL
LIN {X 0,Y 91.584,Z 432.822,A -85,B 0,C 180,E1 -27946.318,E2 -27946.318} C_VEL
LIN {X 0,Y 85.483,Z 438.338,A -85,B 0,C 180,E1 -27951.931,E2 -27951.931} C_VEL
LIN {X 0,Y 80.185,Z 442.662,A -85,B 0,C 180,E1 -27958.272,E2 -27958.272} C_VEL
LIN {X 0,Y 77.247,Z 444.932,A -85,B 0,C 180,E1 -27962.941,E2 -27962.941} C_VEL
LIN {X 0,Y 74.83,Z 446.777,A -85,B 0,C 180,E1 -27967.934,E2 -27967.934} C_VEL
LIN {X 0,Y 72.957,Z 448.175,A -85,B 0,C 180,E1 -27973.202,E2 -27973.202} C_VEL
LIN {X 0,Y 71.066,Z 449.53,A -85,B 0,C 180,E1 -27981.472,E2 -27981.472} C_VEL
LIN {X 0,Y 70.458,Z 449.987,A -85,B 0,C 180,E1 -27990,E2 -27990} C_VEL
LIN {X 0,Y 71.587,Z 449.198,A -85,B 0,C 180,E1 -28001.324,E2 -28001.324} C_VEL
LIN {X 0,Y 72.905,Z 448.234,A -85,B 0,C 180,E1 -28006.81,E2 -28006.81} C_VEL
LIN {X 0,Y 74.772,Z 446.87,A -85,B 0,C 180,E1 -28012.084,E2 -28012.084} C_VEL
LIN {X 0,Y 78.604,Z 443.998,A -85,B 0,C 180,E1 -28019.456,E2 -28019.456} C_VEL
LIN {X 0,Y 83.576,Z 440.083,A -85,B 0,C 180,E1 -28026.06,E2 -28026.06} C_VEL
LIN {X 0,Y 89.4,Z 435.005,A -85,B 0,C 180,E1 -28031.929,E2 -28031.929} C_VEL
LIN {X 0,Y 96.032,Z 428.589,A -85,B 0,C 180,E1 -28037.041,E2 -28037.041} C_VEL
LIN {X 0,Y 103.321,Z 420.601,A -85,B 0,C 180,E1 -28041.466,E2 -28041.466} C_VEL
LIN {X 0,Y 108.451,Z 413.939,A -85,B 0,C 180,E1 -28044.321,E2 -28044.321} C_VEL
LIN {X 0,Y 108.287,Z 413.002,A -85,B 0,C 180,E1 -28045.396,E2 -28045.396} C_VEL
LIN {X 0,Y 101.81,Z 415.532,A -85,B 0,C 180,E1 -28048.82,E2 -28048.82} C_VEL
LIN {X 0,Y 98.916,Z 416.998,A -85,B 0,C 180,E1 -28050.175,E2 -28050.175} C_VEL
LIN {X 0,Y 89.759,Z 420.748,A -85,B 0,C 180,E1 -28056.952,E2 -28056.952} C_VEL
LIN {X 0,Y 82.771,Z 423.741,A -85,B 0,C 180,E1 -28065.242,E2 -28065.242} C_VEL
LIN {X 0,Y 77.397,Z 426.999,A -85,B 0,C 180,E1 -28077.263,E2 -28077.263} C_VEL
LIN {X 0,Y 76.384,Z 431.392,A -85,B 0,C 180,E1 -28096.023,E2 -28096.023} C_VEL
LIN {X 0,Y 78.059,Z 432.23,A -85,B 0,C 180,E1 -28101.108,E2 -28101.108} C_VEL
LIN {X 0,Y 79.398,Z 433.763,A -85,B 0,C 180,E1 -28106.268,E2 -28106.268} C_VEL
LIN {X 0,Y 82.091,Z 434.7,A -85,B 0,C 180,E1 -28110.909,E2 -28110.909} C_VEL
LIN {X 0,Y 84.491,Z 434.927,A -85,B 0,C 180,E1 -28113.44,E2 -28113.44} C_VEL
LIN {X 0,Y 93.929,Z 442.477,A -85,B 0,C 180,E1 -28122.33,E2 -28122.33} C_VEL
LIN {X 0,Y 94.592,Z 443.108,A -85,B 0,C 180,E1 -28124.132,E2 -28124.132} C_VEL
LIN {X 0,Y 90.687,Z 441.727,A -85,B 0,C 180,E1 -28127.304,E2 -28127.304} C_VEL
LIN {X 0,Y 84.861,Z 446.282,A -85,B 0,C 180,E1 -28131.601,E2 -28131.601} C_VEL
LIN {X 0,Y 78.994,Z 450.655,A -85,B 0,C 180,E1 -28137.737,E2 -28137.737} C_VEL
LIN {X 0,Y 75.94,Z 452.98,A -85,B 0,C 180,E1 -28142.436,E2 -28142.436} C_VEL
LIN {X 0,Y 73.532,Z 454.883,A -85,B 0,C 180,E1 -28147.523,E2 -28147.523} C_VEL
LIN {X 0,Y 71.774,Z 456.324,A -85,B 0,C 180,E1 -28152.917,E2 -28152.917} C_VEL
LIN {X 0,Y 70.165,Z 457.99,A -85,B 0,C 180,E1 -28164.251,E2 -28164.251} C_VEL
LIN {X 0,Y 70.28,Z 458.227,A -85,B 0,C 180,E1 -28170,E2 -28170} C_VEL
LIN {X 0,Y 70.046,Z 457.966,A -85,B 0,C 180,E1 -28175.758,E2 -28175.758} C_VEL
LIN {X 0,Y 71.327,Z 456.258,A -85,B 0,C 180,E1 -28187.193,E2 -28187.193} C_VEL
LIN {X 0,Y 72.912,Z 454.783,A -85,B 0,C 180,E1 -28192.679,E2 -28192.679} C_VEL
LIN {X 0,Y 76.552,Z 451.757,A -85,B 0,C 180,E1 -28200.327,E2 -28200.327} C_VEL
LIN {X 0,Y 81.608,Z 447.687,A -85,B 0,C 180,E1 -28207.073,E2 -28207.073} C_VEL
LIN {X 0,Y 87.848,Z 442.455,A -85,B 0,C 180,E1 -28212.845,E2 -28212.845} C_VEL
LIN {X 0,Y 95.19,Z 435.91,A -85,B 0,C 180,E1 -28217.588,E2 -28217.588} C_VEL
LIN {X 0,Y 95.544,Z 434.932,A -85,B 0,C 180,E1 -28218.546,E2 -28218.546} C_VEL
LIN {X 0,Y 91.716,Z 433.93,A -85,B 0,C 180,E1 -28222.192,E2 -28222.192} C_VEL
LIN {X 0,Y 87.836,Z 433.303,A -85,B 0,C 180,E1 -28225.938,E2 -28225.938} C_VEL
LIN {X 0,Y 84.684,Z 432.393,A -85,B 0,C 180,E1 -28230.136,E2 -28230.136} C_VEL
LIN {X 0,Y 82.516,Z 431.051,A -85,B 0,C 180,E1 -28234.795,E2 -28234.795} C_VEL
LIN {X 0,Y 80.242,Z 430.262,A -85,B 0,C 180,E1 -28239.492,E2 -28239.492} C_VEL
LIN {X 0,Y 78.546,Z 426.621,A -85,B 0,C 180,E1 -28254.867,E2 -28254.867} C_VEL
LIN {X 0,Y 79.452,Z 425.189,A -85,B 0,C 180,E1 -28260,E2 -28260} C_VEL
LIN {X 0,Y 81.347,Z 423.449,A -85,B 0,C 180,E1 -28264.957,E2 -28264.957} C_VEL
LIN {X 0,Y 86.24,Z 420.312,A -85,B 0,C 180,E1 -28274.151,E2 -28274.151} C_VEL
LIN {X 0,Y 93.343,Z 416.818,A -85,B 0,C 180,E1 -28282.115,E2 -28282.115} C_VEL
LIN {X 0,Y 100.35,Z 413.33,A -85,B 0,C 180,E1 -28287.08,E2 -28287.08} C_VEL
LIN {X 0,Y 107.74,Z 409.949,A -85,B 0,C 180,E1 -28291.457,E2 -28291.457} C_VEL
LIN {X 0,Y 110.024,Z 408.639,A -85,B 0,C 180,E1 -28292.333,E2 -28292.333} C_VEL
LIN {X 0,Y 109.947,Z 410.256,A -85,B 0,C 180,E1 -28293.8,E2 -28293.8} C_VEL
LIN {X 0,Y 108.612,Z 413.367,A -85,B 0,C 180,E1 -28295.617,E2 -28295.617} C_VEL
LIN {X 0,Y 105.149,Z 418.102,A -85,B 0,C 180,E1 -28297.605,E2 -28297.605} C_VEL
LIN {X 0,Y 102.615,Z 420.76,A -85,B 0,C 180,E1 -28298.475,E2 -28298.475} C_VEL
LIN {X 0,Y 97.337,Z 424.842,A -85,B 0,C 180,E1 -28299.146,E2 -28299.146} C_VEL
LIN {X 0,Y 91.913,Z 428.645,A -85,B 0,C 180,E1 -28299.985,E2 -28299.985} C_VEL
LIN {X 0,Y 89.203,Z 430.846,A -85,B 0,C 180,E1 -28301.199,E2 -28301.199} C_VEL
LIN {X 0,Y 82.159,Z 437.037,A -85,B 0,C 180,E1 -28306.817,E2 -28306.817} C_VEL
LIN {X 0,Y 76.059,Z 441.753,A -85,B 0,C 180,E1 -28313.086,E2 -28313.086} C_VEL
LIN {X 0,Y 71.022,Z 445.346,A -85,B 0,C 180,E1 -28320.345,E2 -28320.345} C_VEL
LIN {X 0,Y 68.311,Z 447.193,A -85,B 0,C 180,E1 -28325.699,E2 -28325.699} C_VEL
LIN {X 0,Y 66.208,Z 448.589,A -85,B 0,C 180,E1 -28331.431,E2 -28331.431} C_VEL
LIN {X 0,Y 63.836,Z 450.072,A -85,B 0,C 180,E1 -28342.25,E2 -28342.25} C_VEL
LIN {X 0,Y 63.381,Z 450.402,A -85,B 0,C 180,E1 -28350,E2 -28350} C_VEL
LIN {X 0,Y 63.836,Z 450.097,A -85,B 0,C 180,E1 -28357.75,E2 -28357.75} C_VEL
LIN {X 0,Y 66.143,Z 448.649,A -85,B 0,C 180,E1 -28368.588,E2 -28368.588} C_VEL
LIN {X 0,Y 68.246,Z 447.285,A -85,B 0,C 180,E1 -28374.326,E2 -28374.326} C_VEL
LIN {X 0,Y 72.52,Z 444.411,A -85,B 0,C 180,E1 -28382.209,E2 -28382.209} C_VEL
